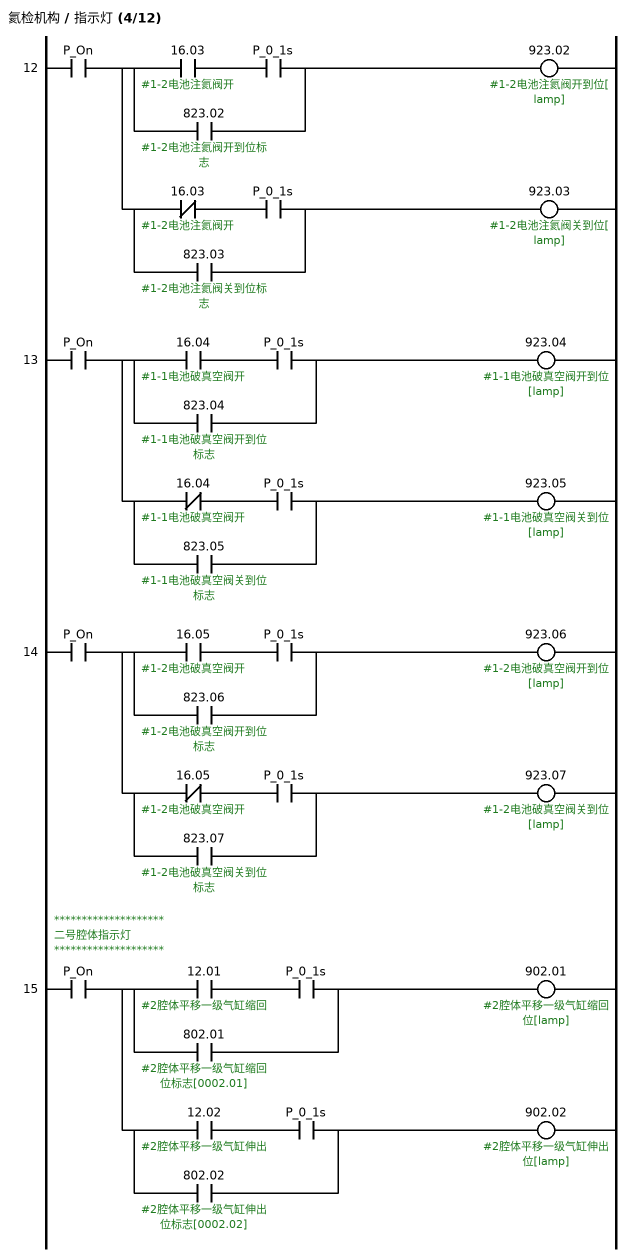
; [picture p360: 氦检机构 / 指示灯, rungs 12-15]
; rung 12
LD P_On
OUT TR0
LD 16.03  ; #1-2电池注氦阀开
AND P_0_1s
OR 823.02  ; #1-2电池注氦阀开到位标志
ANDLD
OUT 923.02  ; #1-2电池注氦阀开到位[lamp]
LD TR0
LDNOT 16.03  ; #1-2电池注氦阀开
AND P_0_1s
OR 823.03  ; #1-2电池注氦阀关到位标志
ANDLD
OUT 923.03  ; #1-2电池注氦阀关到位[lamp]
; rung 13
LD P_On
OUT TR0
LD 16.04  ; #1-1电池破真空阀开
AND P_0_1s
OR 823.04  ; #1-1电池破真空阀开到位标志
ANDLD
OUT 923.04  ; #1-1电池破真空阀开到位[lamp]
LD TR0
LDNOT 16.04  ; #1-1电池破真空阀开
AND P_0_1s
OR 823.05  ; #1-1电池破真空阀关到位标志
ANDLD
OUT 923.05  ; #1-1电池破真空阀关到位[lamp]
; rung 14
LD P_On
OUT TR0
LD 16.05  ; #1-2电池破真空阀开
AND P_0_1s
OR 823.06  ; #1-2电池破真空阀开到位标志
ANDLD
OUT 923.06  ; #1-2电池破真空阀开到位[lamp]
LD TR0
LDNOT 16.05  ; #1-2电池破真空阀开
AND P_0_1s
OR 823.07  ; #1-2电池破真空阀关到位标志
ANDLD
OUT 923.07  ; #1-2电池破真空阀关到位[lamp]
; rung 15: ******************** / 二号腔体指示灯 / ********************
LD P_On
OUT TR0
LD 12.01  ; #2腔体平移一级气缸缩回
AND P_0_1s
OR 802.01  ; #2腔体平移一级气缸缩回位标志[0002.01]
ANDLD
OUT 902.01  ; #2腔体平移一级气缸缩回位[lamp]
LD TR0
LD 12.02  ; #2腔体平移一级气缸伸出
AND P_0_1s
OR 802.02  ; #2腔体平移一级气缸伸出位标志[0002.02]
ANDLD
OUT 902.02  ; #2腔体平移一级气缸伸出位[lamp]

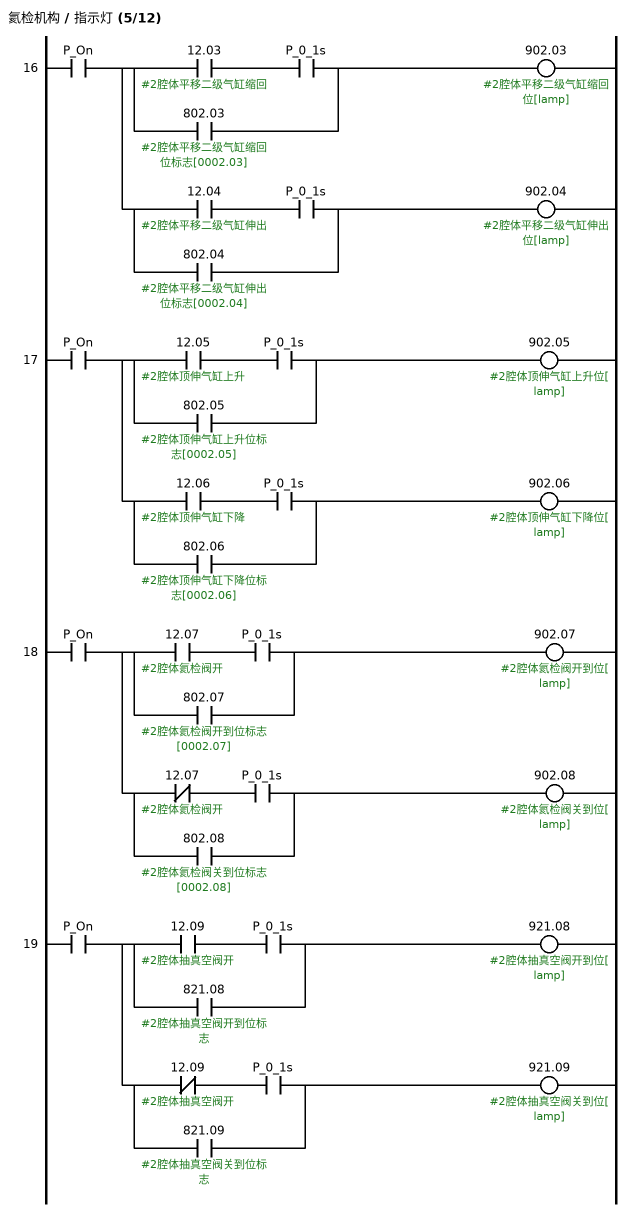
; rung 16
LD P_On
OUT TR0
LD 12.03  ; #2腔体平移二级气缸缩回
AND P_0_1s
OR 802.03  ; #2腔体平移二级气缸缩回位标志[0002.03]
ANDLD
OUT 902.03  ; #2腔体平移二级气缸缩回位[lamp]
LD TR0
LD 12.04  ; #2腔体平移二级气缸伸出
AND P_0_1s
OR 802.04  ; #2腔体平移二级气缸伸出位标志[0002.04]
ANDLD
OUT 902.04  ; #2腔体平移二级气缸伸出位[lamp]
; rung 17
LD P_On
OUT TR0
LD 12.05  ; #2腔体顶伸气缸上升
AND P_0_1s
OR 802.05  ; #2腔体顶伸气缸上升位标志[0002.05]
ANDLD
OUT 902.05  ; #2腔体顶伸气缸上升位[lamp]
LD TR0
LD 12.06  ; #2腔体顶伸气缸下降
AND P_0_1s
OR 802.06  ; #2腔体顶伸气缸下降位标志[0002.06]
ANDLD
OUT 902.06  ; #2腔体顶伸气缸下降位[lamp]
; rung 18
LD P_On
OUT TR0
LD 12.07  ; #2腔体氦检阀开
AND P_0_1s
OR 802.07  ; #2腔体氦检阀开到位标志[0002.07]
ANDLD
OUT 902.07  ; #2腔体氦检阀开到位[lamp]
LD TR0
LDNOT 12.07  ; #2腔体氦检阀开
AND P_0_1s
OR 802.08  ; #2腔体氦检阀关到位标志[0002.08]
ANDLD
OUT 902.08  ; #2腔体氦检阀关到位[lamp]
; rung 19
LD P_On
OUT TR0
LD 12.09  ; #2腔体抽真空阀开
AND P_0_1s
OR 821.08  ; #2腔体抽真空阀开到位标志
ANDLD
OUT 921.08  ; #2腔体抽真空阀开到位[lamp]
LD TR0
LDNOT 12.09  ; #2腔体抽真空阀开
AND P_0_1s
OR 821.09  ; #2腔体抽真空阀关到位标志
ANDLD
OUT 921.09  ; #2腔体抽真空阀关到位[lamp]

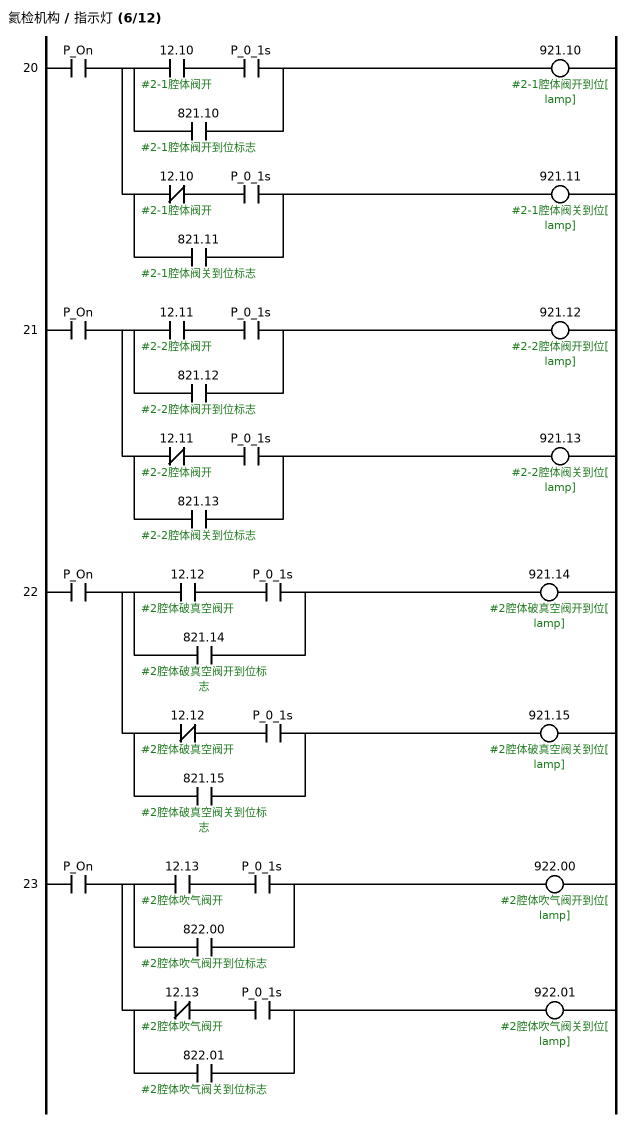
; rung 20
LD P_On
OUT TR0
LD 12.10  ; #2-1腔体阀开
AND P_0_1s
OR 821.10  ; #2-1腔体阀开到位标志
ANDLD
OUT 921.10  ; #2-1腔体阀开到位[lamp]
LD TR0
LDNOT 12.10  ; #2-1腔体阀开
AND P_0_1s
OR 821.11  ; #2-1腔体阀关到位标志
ANDLD
OUT 921.11  ; #2-1腔体阀关到位[lamp]
; rung 21
LD P_On
OUT TR0
LD 12.11  ; #2-2腔体阀开
AND P_0_1s
OR 821.12  ; #2-2腔体阀开到位标志
ANDLD
OUT 921.12  ; #2-2腔体阀开到位[lamp]
LD TR0
LDNOT 12.11  ; #2-2腔体阀开
AND P_0_1s
OR 821.13  ; #2-2腔体阀关到位标志
ANDLD
OUT 921.13  ; #2-2腔体阀关到位[lamp]
; rung 22
LD P_On
OUT TR0
LD 12.12  ; #2腔体破真空阀开
AND P_0_1s
OR 821.14  ; #2腔体破真空阀开到位标志
ANDLD
OUT 921.14  ; #2腔体破真空阀开到位[lamp]
LD TR0
LDNOT 12.12  ; #2腔体破真空阀开
AND P_0_1s
OR 821.15  ; #2腔体破真空阀关到位标志
ANDLD
OUT 921.15  ; #2腔体破真空阀关到位[lamp]
; rung 23
LD P_On
OUT TR0
LD 12.13  ; #2腔体吹气阀开
AND P_0_1s
OR 822.00  ; #2腔体吹气阀开到位标志
ANDLD
OUT 922.00  ; #2腔体吹气阀开到位[lamp]
LD TR0
LDNOT 12.13  ; #2腔体吹气阀开
AND P_0_1s
OR 822.01  ; #2腔体吹气阀关到位标志
ANDLD
OUT 922.01  ; #2腔体吹气阀关到位[lamp]

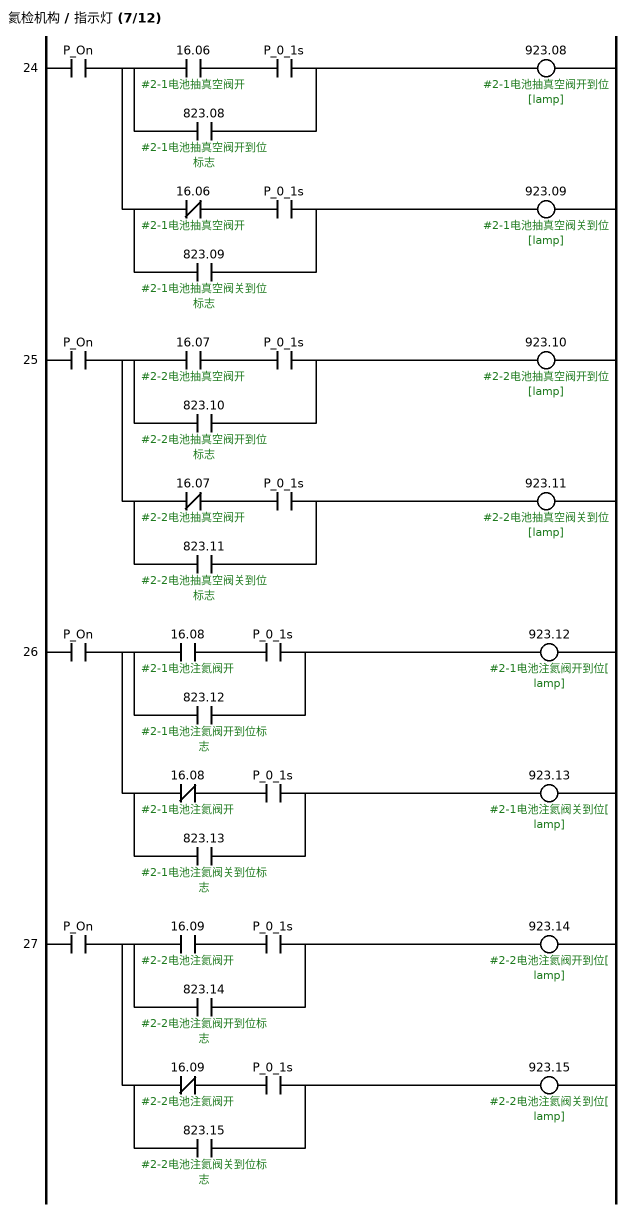
; rung 24
LD P_On
OUT TR0
LD 16.06  ; #2-1电池抽真空阀开
AND P_0_1s
OR 823.08  ; #2-1电池抽真空阀开到位标志
ANDLD
OUT 923.08  ; #2-1电池抽真空阀开到位[lamp]
LD TR0
LDNOT 16.06  ; #2-1电池抽真空阀开
AND P_0_1s
OR 823.09  ; #2-1电池抽真空阀关到位标志
ANDLD
OUT 923.09  ; #2-1电池抽真空阀关到位[lamp]
; rung 25
LD P_On
OUT TR0
LD 16.07  ; #2-2电池抽真空阀开
AND P_0_1s
OR 823.10  ; #2-2电池抽真空阀开到位标志
ANDLD
OUT 923.10  ; #2-2电池抽真空阀开到位[lamp]
LD TR0
LDNOT 16.07  ; #2-2电池抽真空阀开
AND P_0_1s
OR 823.11  ; #2-2电池抽真空阀关到位标志
ANDLD
OUT 923.11  ; #2-2电池抽真空阀关到位[lamp]
; rung 26
LD P_On
OUT TR0
LD 16.08  ; #2-1电池注氦阀开
AND P_0_1s
OR 823.12  ; #2-1电池注氦阀开到位标志
ANDLD
OUT 923.12  ; #2-1电池注氦阀开到位[lamp]
LD TR0
LDNOT 16.08  ; #2-1电池注氦阀开
AND P_0_1s
OR 823.13  ; #2-1电池注氦阀关到位标志
ANDLD
OUT 923.13  ; #2-1电池注氦阀关到位[lamp]
; rung 27
LD P_On
OUT TR0
LD 16.09  ; #2-2电池注氦阀开
AND P_0_1s
OR 823.14  ; #2-2电池注氦阀开到位标志
ANDLD
OUT 923.14  ; #2-2电池注氦阀开到位[lamp]
LD TR0
LDNOT 16.09  ; #2-2电池注氦阀开
AND P_0_1s
OR 823.15  ; #2-2电池注氦阀关到位标志
ANDLD
OUT 923.15  ; #2-2电池注氦阀关到位[lamp]

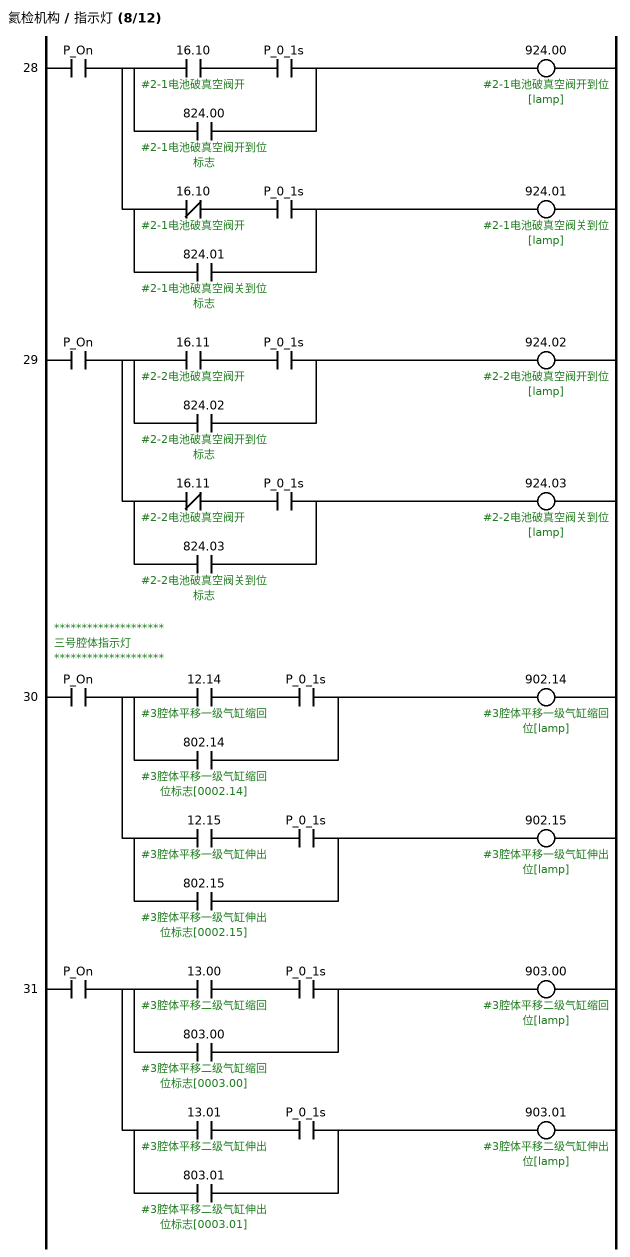
; rung 28
LD P_On
OUT TR0
LD 16.10  ; #2-1电池破真空阀开
AND P_0_1s
OR 824.00  ; #2-1电池破真空阀开到位标志
ANDLD
OUT 924.00  ; #2-1电池破真空阀开到位[lamp]
LD TR0
LDNOT 16.10  ; #2-1电池破真空阀开
AND P_0_1s
OR 824.01  ; #2-1电池破真空阀关到位标志
ANDLD
OUT 924.01  ; #2-1电池破真空阀关到位[lamp]
; rung 29
LD P_On
OUT TR0
LD 16.11  ; #2-2电池破真空阀开
AND P_0_1s
OR 824.02  ; #2-2电池破真空阀开到位标志
ANDLD
OUT 924.02  ; #2-2电池破真空阀开到位[lamp]
LD TR0
LDNOT 16.11  ; #2-2电池破真空阀开
AND P_0_1s
OR 824.03  ; #2-2电池破真空阀关到位标志
ANDLD
OUT 924.03  ; #2-2电池破真空阀关到位[lamp]
; rung 30: ******************** / 三号腔体指示灯 / ********************
LD P_On
OUT TR0
LD 12.14  ; #3腔体平移一级气缸缩回
AND P_0_1s
OR 802.14  ; #3腔体平移一级气缸缩回位标志[0002.14]
ANDLD
OUT 902.14  ; #3腔体平移一级气缸缩回位[lamp]
LD TR0
LD 12.15  ; #3腔体平移一级气缸伸出
AND P_0_1s
OR 802.15  ; #3腔体平移一级气缸伸出位标志[0002.15]
ANDLD
OUT 902.15  ; #3腔体平移一级气缸伸出位[lamp]
; rung 31
LD P_On
OUT TR0
LD 13.00  ; #3腔体平移二级气缸缩回
AND P_0_1s
OR 803.00  ; #3腔体平移二级气缸缩回位标志[0003.00]
ANDLD
OUT 903.00  ; #3腔体平移二级气缸缩回位[lamp]
LD TR0
LD 13.01  ; #3腔体平移二级气缸伸出
AND P_0_1s
OR 803.01  ; #3腔体平移二级气缸伸出位标志[0003.01]
ANDLD
OUT 903.01  ; #3腔体平移二级气缸伸出位[lamp]

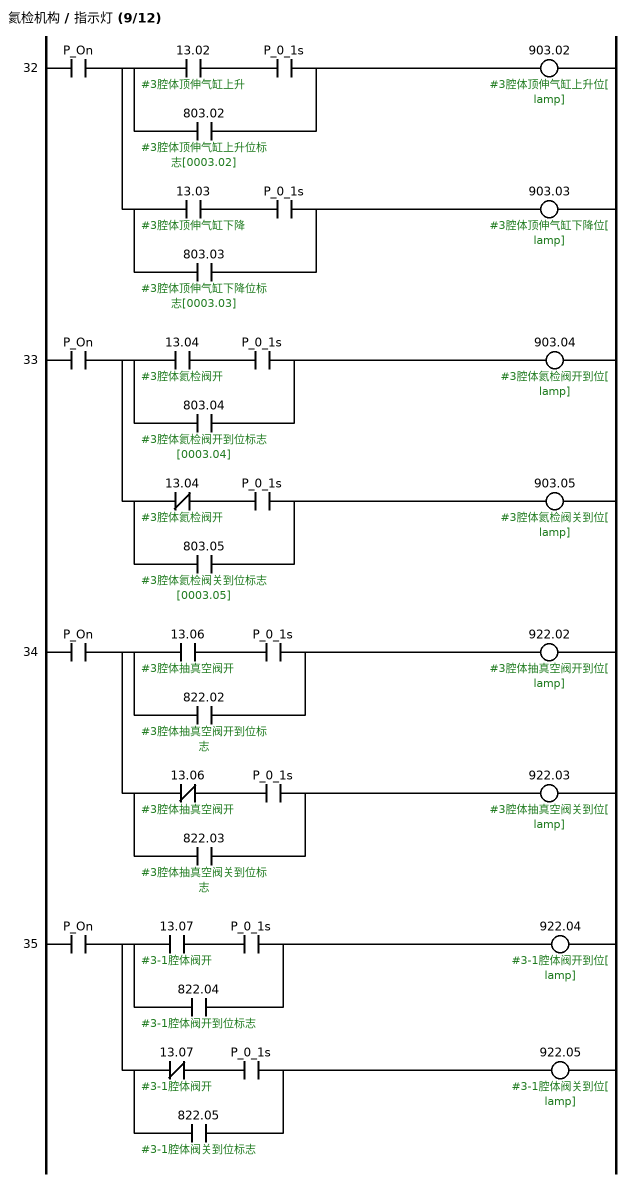
; rung 32
LD P_On
OUT TR0
LD 13.02  ; #3腔体顶伸气缸上升
AND P_0_1s
OR 803.02  ; #3腔体顶伸气缸上升位标志[0003.02]
ANDLD
OUT 903.02  ; #3腔体顶伸气缸上升位[lamp]
LD TR0
LD 13.03  ; #3腔体顶伸气缸下降
AND P_0_1s
OR 803.03  ; #3腔体顶伸气缸下降位标志[0003.03]
ANDLD
OUT 903.03  ; #3腔体顶伸气缸下降位[lamp]
; rung 33
LD P_On
OUT TR0
LD 13.04  ; #3腔体氦检阀开
AND P_0_1s
OR 803.04  ; #3腔体氦检阀开到位标志[0003.04]
ANDLD
OUT 903.04  ; #3腔体氦检阀开到位[lamp]
LD TR0
LDNOT 13.04  ; #3腔体氦检阀开
AND P_0_1s
OR 803.05  ; #3腔体氦检阀关到位标志[0003.05]
ANDLD
OUT 903.05  ; #3腔体氦检阀关到位[lamp]
; rung 34
LD P_On
OUT TR0
LD 13.06  ; #3腔体抽真空阀开
AND P_0_1s
OR 822.02  ; #3腔体抽真空阀开到位标志
ANDLD
OUT 922.02  ; #3腔体抽真空阀开到位[lamp]
LD TR0
LDNOT 13.06  ; #3腔体抽真空阀开
AND P_0_1s
OR 822.03  ; #3腔体抽真空阀关到位标志
ANDLD
OUT 922.03  ; #3腔体抽真空阀关到位[lamp]
; rung 35
LD P_On
OUT TR0
LD 13.07  ; #3-1腔体阀开
AND P_0_1s
OR 822.04  ; #3-1腔体阀开到位标志
ANDLD
OUT 922.04  ; #3-1腔体阀开到位[lamp]
LD TR0
LDNOT 13.07  ; #3-1腔体阀开
AND P_0_1s
OR 822.05  ; #3-1腔体阀关到位标志
ANDLD
OUT 922.05  ; #3-1腔体阀关到位[lamp]

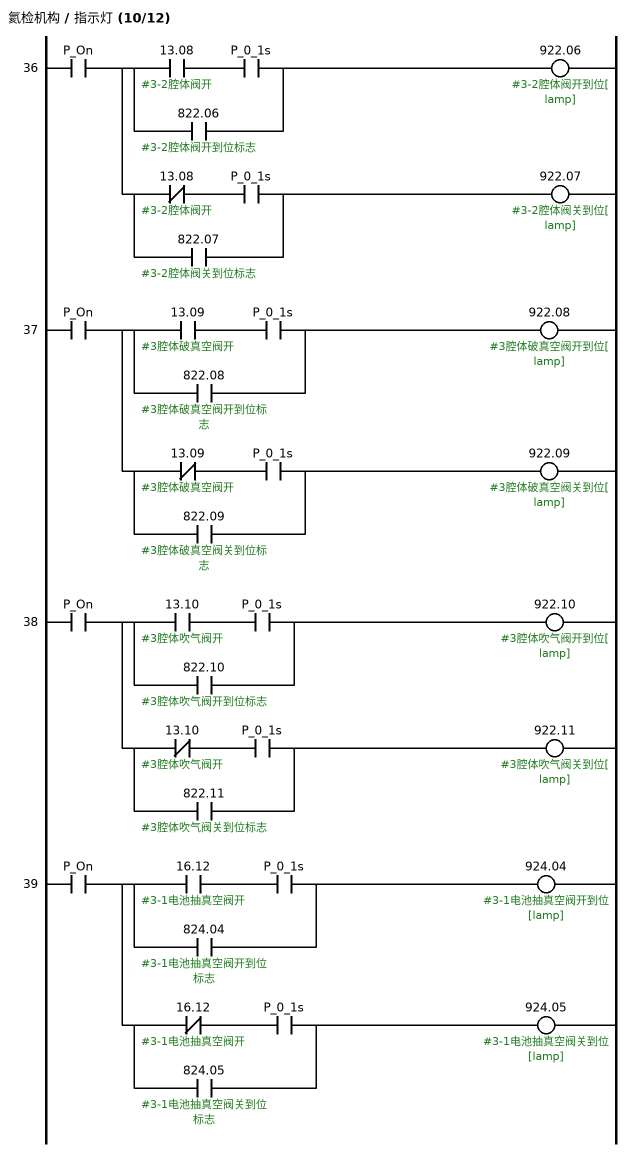
; rung 36
LD P_On
OUT TR0
LD 13.08  ; #3-2腔体阀开
AND P_0_1s
OR 822.06  ; #3-2腔体阀开到位标志
ANDLD
OUT 922.06  ; #3-2腔体阀开到位[lamp]
LD TR0
LDNOT 13.08  ; #3-2腔体阀开
AND P_0_1s
OR 822.07  ; #3-2腔体阀关到位标志
ANDLD
OUT 922.07  ; #3-2腔体阀关到位[lamp]
; rung 37
LD P_On
OUT TR0
LD 13.09  ; #3腔体破真空阀开
AND P_0_1s
OR 822.08  ; #3腔体破真空阀开到位标志
ANDLD
OUT 922.08  ; #3腔体破真空阀开到位[lamp]
LD TR0
LDNOT 13.09  ; #3腔体破真空阀开
AND P_0_1s
OR 822.09  ; #3腔体破真空阀关到位标志
ANDLD
OUT 922.09  ; #3腔体破真空阀关到位[lamp]
; rung 38
LD P_On
OUT TR0
LD 13.10  ; #3腔体吹气阀开
AND P_0_1s
OR 822.10  ; #3腔体吹气阀开到位标志
ANDLD
OUT 922.10  ; #3腔体吹气阀开到位[lamp]
LD TR0
LDNOT 13.10  ; #3腔体吹气阀开
AND P_0_1s
OR 822.11  ; #3腔体吹气阀关到位标志
ANDLD
OUT 922.11  ; #3腔体吹气阀关到位[lamp]
; rung 39
LD P_On
OUT TR0
LD 16.12  ; #3-1电池抽真空阀开
AND P_0_1s
OR 824.04  ; #3-1电池抽真空阀开到位标志
ANDLD
OUT 924.04  ; #3-1电池抽真空阀开到位[lamp]
LD TR0
LDNOT 16.12  ; #3-1电池抽真空阀开
AND P_0_1s
OR 824.05  ; #3-1电池抽真空阀关到位标志
ANDLD
OUT 924.05  ; #3-1电池抽真空阀关到位[lamp]

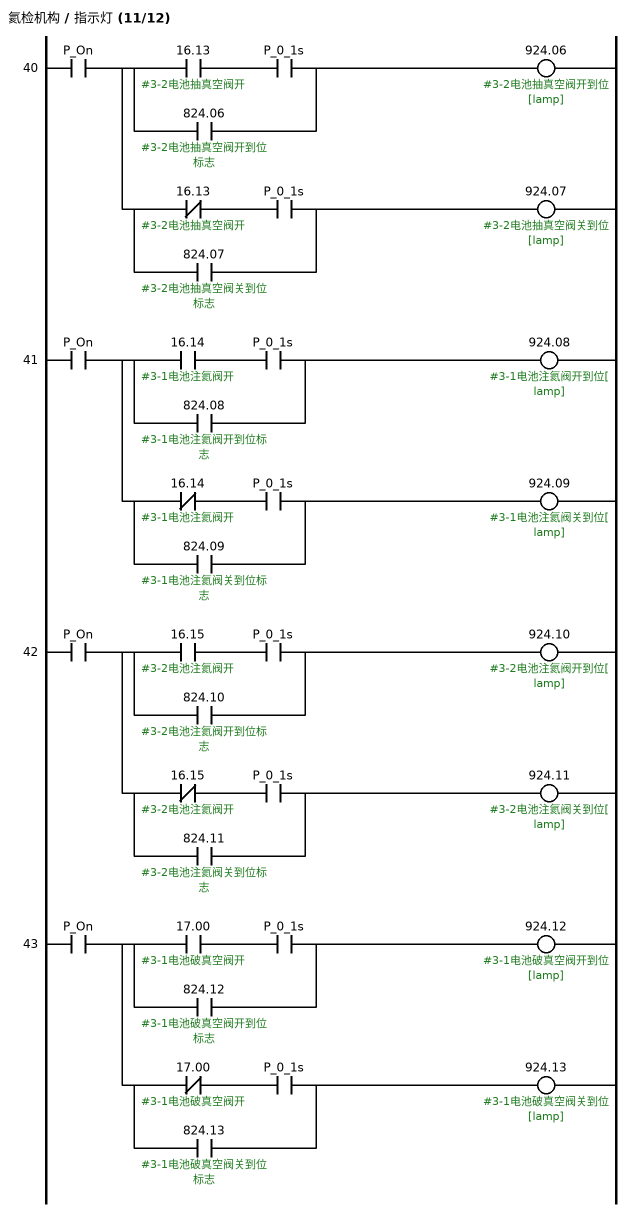
; rung 40
LD P_On
OUT TR0
LD 16.13  ; #3-2电池抽真空阀开
AND P_0_1s
OR 824.06  ; #3-2电池抽真空阀开到位标志
ANDLD
OUT 924.06  ; #3-2电池抽真空阀开到位[lamp]
LD TR0
LDNOT 16.13  ; #3-2电池抽真空阀开
AND P_0_1s
OR 824.07  ; #3-2电池抽真空阀关到位标志
ANDLD
OUT 924.07  ; #3-2电池抽真空阀关到位[lamp]
; rung 41
LD P_On
OUT TR0
LD 16.14  ; #3-1电池注氦阀开
AND P_0_1s
OR 824.08  ; #3-1电池注氦阀开到位标志
ANDLD
OUT 924.08  ; #3-1电池注氦阀开到位[lamp]
LD TR0
LDNOT 16.14  ; #3-1电池注氦阀开
AND P_0_1s
OR 824.09  ; #3-1电池注氦阀关到位标志
ANDLD
OUT 924.09  ; #3-1电池注氦阀关到位[lamp]
; rung 42
LD P_On
OUT TR0
LD 16.15  ; #3-2电池注氦阀开
AND P_0_1s
OR 824.10  ; #3-2电池注氦阀开到位标志
ANDLD
OUT 924.10  ; #3-2电池注氦阀开到位[lamp]
LD TR0
LDNOT 16.15  ; #3-2电池注氦阀开
AND P_0_1s
OR 824.11  ; #3-2电池注氦阀关到位标志
ANDLD
OUT 924.11  ; #3-2电池注氦阀关到位[lamp]
; rung 43
LD P_On
OUT TR0
LD 17.00  ; #3-1电池破真空阀开
AND P_0_1s
OR 824.12  ; #3-1电池破真空阀开到位标志
ANDLD
OUT 924.12  ; #3-1电池破真空阀开到位[lamp]
LD TR0
LDNOT 17.00  ; #3-1电池破真空阀开
AND P_0_1s
OR 824.13  ; #3-1电池破真空阀关到位标志
ANDLD
OUT 924.13  ; #3-1电池破真空阀关到位[lamp]

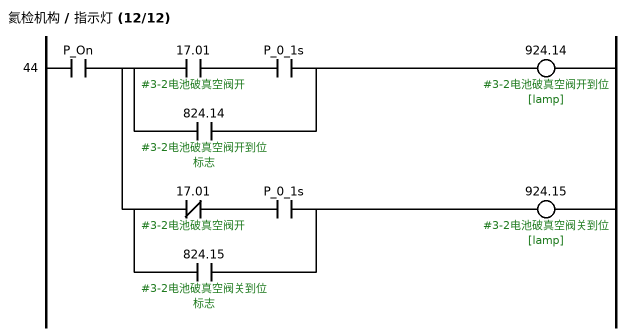
; rung 44
LD P_On
OUT TR0
LD 17.01  ; #3-2电池破真空阀开
AND P_0_1s
OR 824.14  ; #3-2电池破真空阀开到位标志
ANDLD
OUT 924.14  ; #3-2电池破真空阀开到位[lamp]
LD TR0
LDNOT 17.01  ; #3-2电池破真空阀开
AND P_0_1s
OR 824.15  ; #3-2电池破真空阀关到位标志
ANDLD
OUT 924.15  ; #3-2电池破真空阀关到位[lamp]

### Section 外部输出

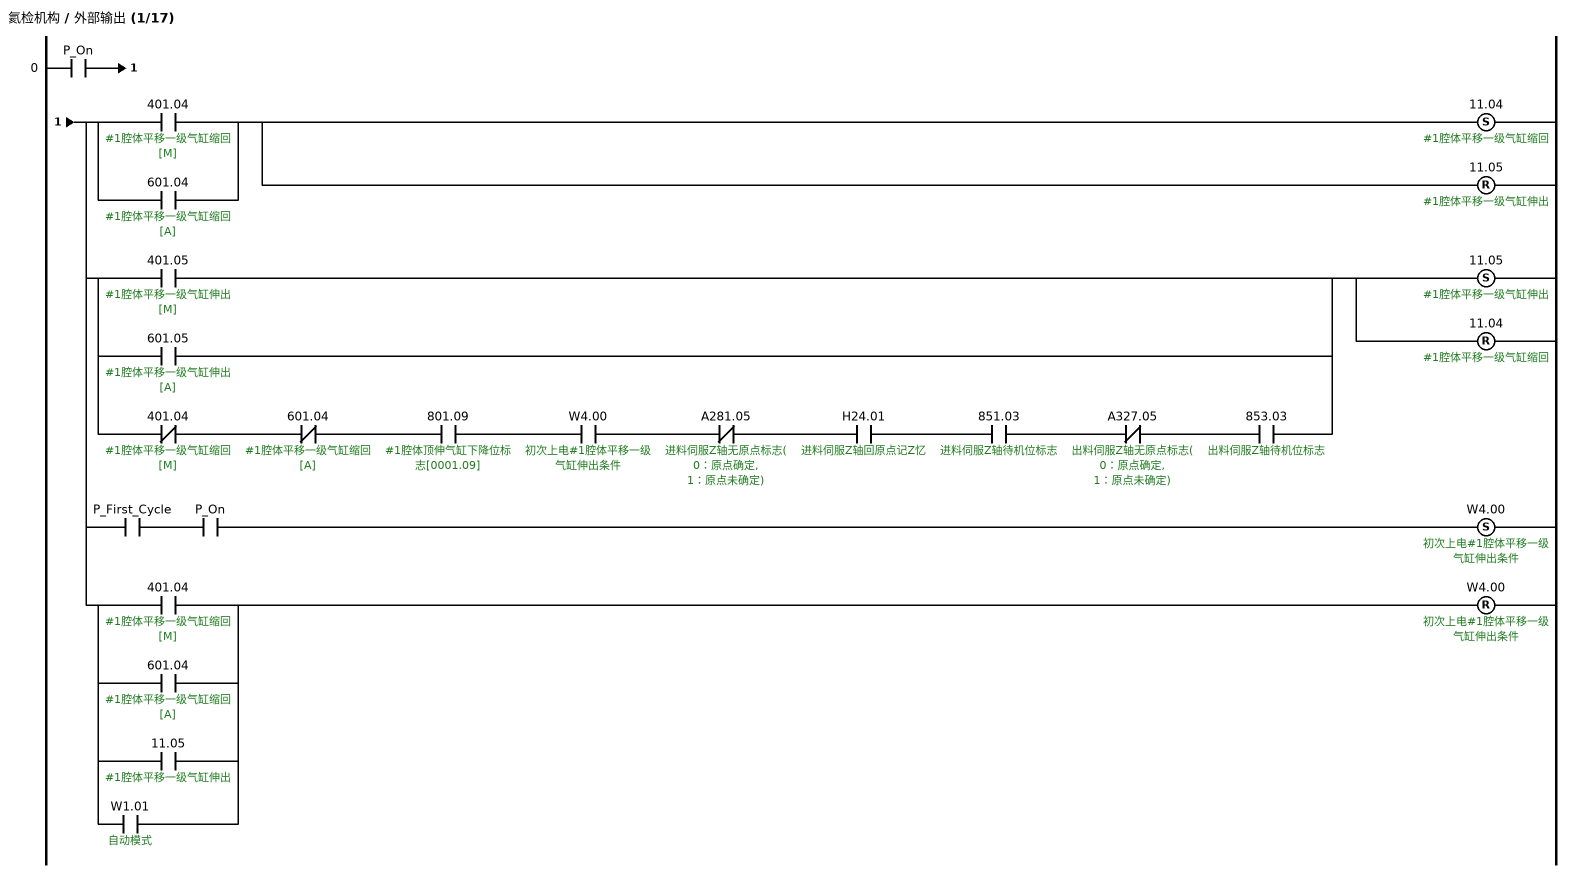
; rung 0
LD P_On
OUT TR0
LD 401.04  ; #1腔体平移一级气缸缩回[M]
OR 601.04  ; #1腔体平移一级气缸缩回[A]
ANDLD
SET 11.04  ; #1腔体平移一级气缸缩回
RSET 11.05  ; #1腔体平移一级气缸伸出
LD TR0
LD 401.05  ; #1腔体平移一级气缸伸出[M]
OR 601.05  ; #1腔体平移一级气缸伸出[A]
LDNOT 401.04  ; #1腔体平移一级气缸缩回[M]
ANDNOT 601.04  ; #1腔体平移一级气缸缩回[A]
AND 801.09  ; #1腔体顶伸气缸下降位标志[0001.09]
AND W4.00  ; 初次上电#1腔体平移一级气缸伸出条件
ANDNOT A281.05  ; 进料伺服Z轴无原点标志(0：原点确定,1：原点未确定)
AND H24.01  ; 进料伺服Z轴回原点记Z忆
AND 851.03  ; 进料伺服Z轴待机位标志
ANDNOT A327.05  ; 出料伺服Z轴无原点标志(0：原点确定,1：原点未确定)
AND 853.03  ; 出料伺服Z轴待机位标志
ORLD
ANDLD
SET 11.05  ; #1腔体平移一级气缸伸出
RSET 11.04  ; #1腔体平移一级气缸缩回
LD TR0
AND P_First_Cycle
AND P_On
SET W4.00  ; 初次上电#1腔体平移一级气缸伸出条件
LD TR0
LD 401.04  ; #1腔体平移一级气缸缩回[M]
OR 601.04  ; #1腔体平移一级气缸缩回[A]
OR 11.05  ; #1腔体平移一级气缸伸出
OR W1.01  ; 自动模式
ANDLD
RSET W4.00  ; 初次上电#1腔体平移一级气缸伸出条件

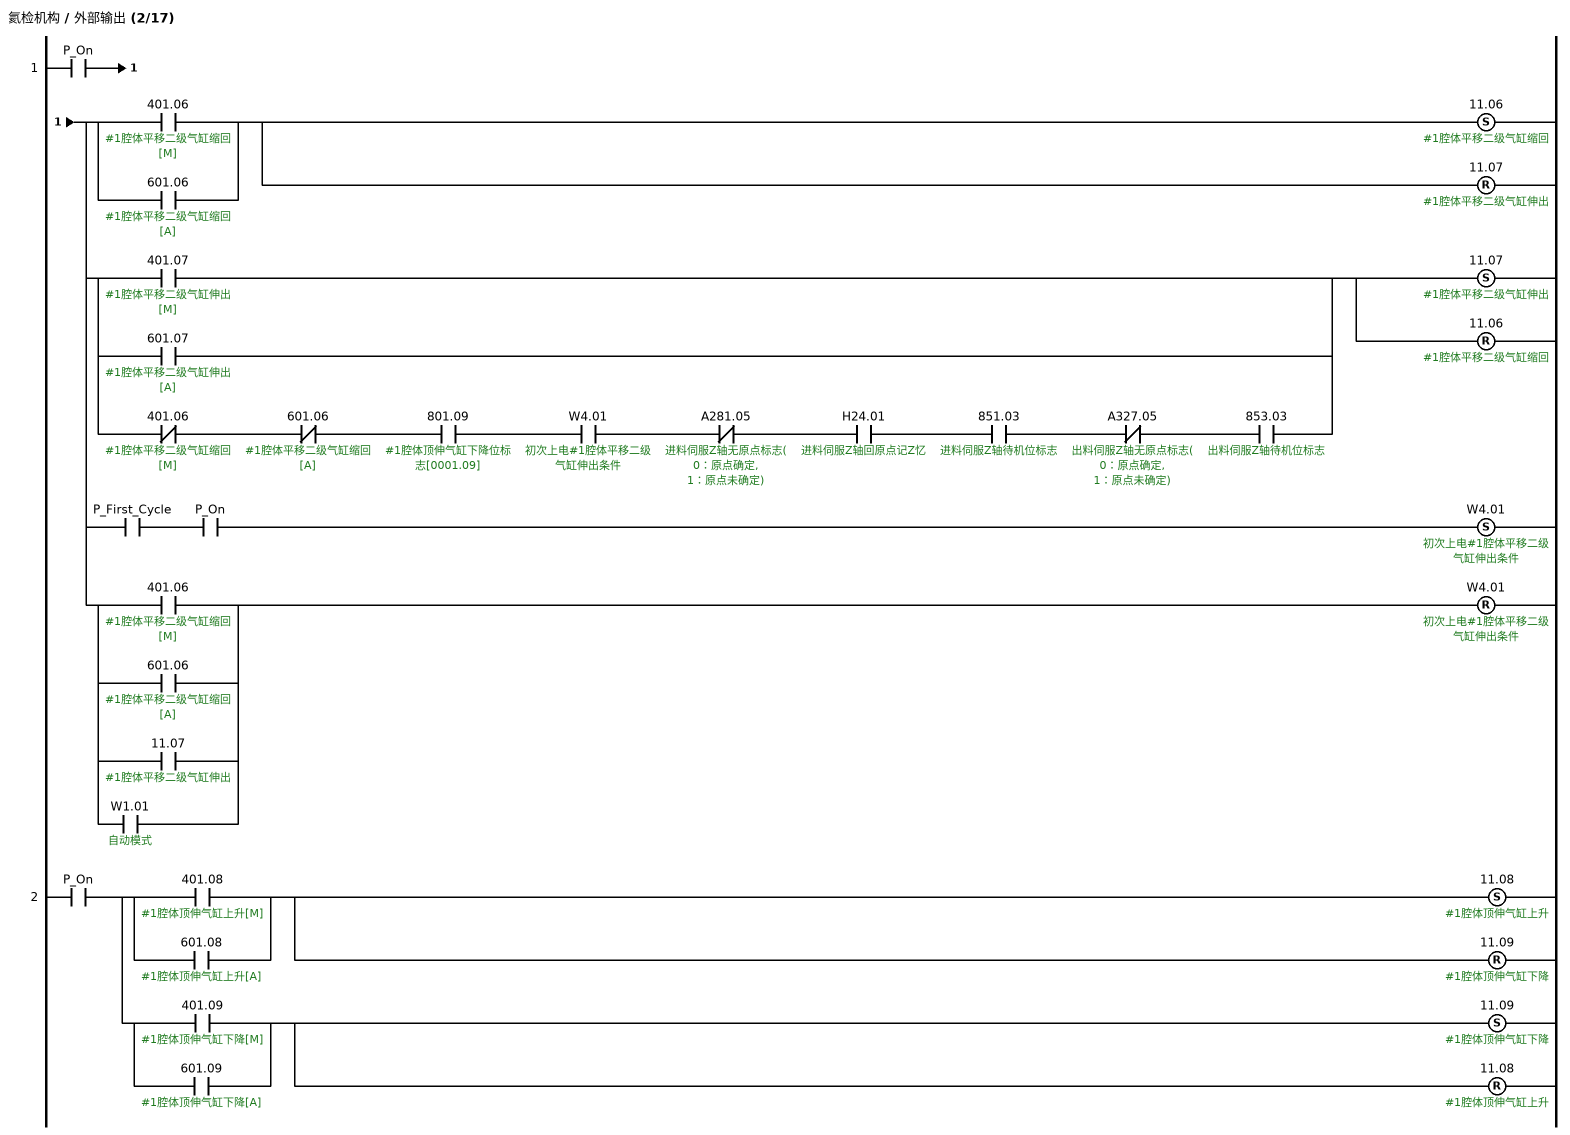
; rung 1
LD P_On
OUT TR0
LD 401.06  ; #1腔体平移二级气缸缩回[M]
OR 601.06  ; #1腔体平移二级气缸缩回[A]
ANDLD
SET 11.06  ; #1腔体平移二级气缸缩回
RSET 11.07  ; #1腔体平移二级气缸伸出
LD TR0
LD 401.07  ; #1腔体平移二级气缸伸出[M]
OR 601.07  ; #1腔体平移二级气缸伸出[A]
LDNOT 401.06  ; #1腔体平移二级气缸缩回[M]
ANDNOT 601.06  ; #1腔体平移二级气缸缩回[A]
AND 801.09  ; #1腔体顶伸气缸下降位标志[0001.09]
AND W4.01  ; 初次上电#1腔体平移二级气缸伸出条件
ANDNOT A281.05  ; 进料伺服Z轴无原点标志(0：原点确定,1：原点未确定)
AND H24.01  ; 进料伺服Z轴回原点记Z忆
AND 851.03  ; 进料伺服Z轴待机位标志
ANDNOT A327.05  ; 出料伺服Z轴无原点标志(0：原点确定,1：原点未确定)
AND 853.03  ; 出料伺服Z轴待机位标志
ORLD
ANDLD
SET 11.07  ; #1腔体平移二级气缸伸出
RSET 11.06  ; #1腔体平移二级气缸缩回
LD TR0
AND P_First_Cycle
AND P_On
SET W4.01  ; 初次上电#1腔体平移二级气缸伸出条件
LD TR0
LD 401.06  ; #1腔体平移二级气缸缩回[M]
OR 601.06  ; #1腔体平移二级气缸缩回[A]
OR 11.07  ; #1腔体平移二级气缸伸出
OR W1.01  ; 自动模式
ANDLD
RSET W4.01  ; 初次上电#1腔体平移二级气缸伸出条件
; rung 2
LD P_On
OUT TR0
LD 401.08  ; #1腔体顶伸气缸上升[M]
OR 601.08  ; #1腔体顶伸气缸上升[A]
ANDLD
SET 11.08  ; #1腔体顶伸气缸上升
RSET 11.09  ; #1腔体顶伸气缸下降
LD TR0
LD 401.09  ; #1腔体顶伸气缸下降[M]
OR 601.09  ; #1腔体顶伸气缸下降[A]
ANDLD
SET 11.09  ; #1腔体顶伸气缸下降
RSET 11.08  ; #1腔体顶伸气缸上升

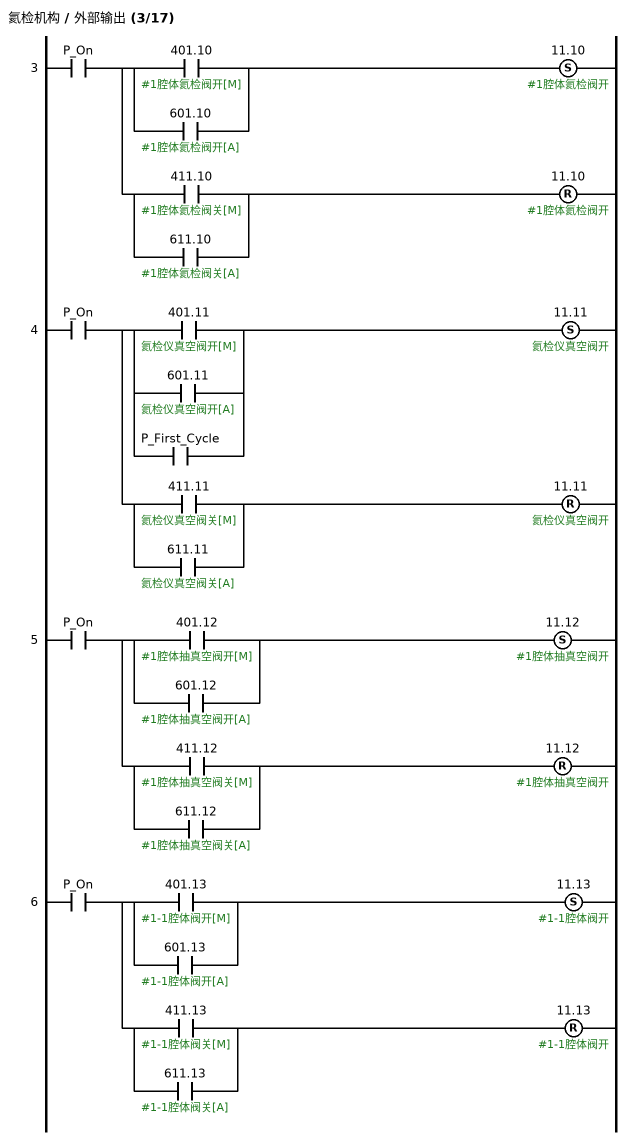
; rung 3
LD P_On
OUT TR0
LD 401.10  ; #1腔体氦检阀开[M]
OR 601.10  ; #1腔体氦检阀开[A]
ANDLD
SET 11.10  ; #1腔体氦检阀开
LD TR0
LD 411.10  ; #1腔体氦检阀关[M]
OR 611.10  ; #1腔体氦检阀关[A]
ANDLD
RSET 11.10  ; #1腔体氦检阀开
; rung 4
LD P_On
OUT TR0
LD 401.11  ; 氦检仪真空阀开[M]
OR 601.11  ; 氦检仪真空阀开[A]
OR P_First_Cycle  // 保证氦检仪开启时能将管路抽成真空状态
ANDLD
SET 11.11  ; 氦检仪真空阀开
LD TR0
LD 411.11  ; 氦检仪真空阀关[M]
OR 611.11  ; 氦检仪真空阀关[A]
ANDLD
RSET 11.11  ; 氦检仪真空阀开
; rung 5
LD P_On
OUT TR0
LD 401.12  ; #1腔体抽真空阀开[M]
OR 601.12  ; #1腔体抽真空阀开[A]
ANDLD
SET 11.12  ; #1腔体抽真空阀开
LD TR0
LD 411.12  ; #1腔体抽真空阀关[M]
OR 611.12  ; #1腔体抽真空阀关[A]
ANDLD
RSET 11.12  ; #1腔体抽真空阀开
; rung 6
LD P_On
OUT TR0
LD 401.13  ; #1-1腔体阀开[M]
OR 601.13  ; #1-1腔体阀开[A]
ANDLD
SET 11.13  ; #1-1腔体阀开
LD TR0
LD 411.13  ; #1-1腔体阀关[M]
OR 611.13  ; #1-1腔体阀关[A]
ANDLD
RSET 11.13  ; #1-1腔体阀开

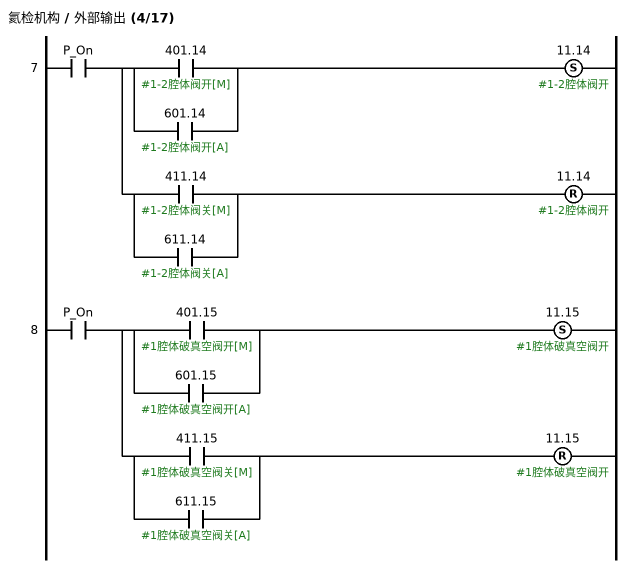
; rung 7
LD P_On
OUT TR0
LD 401.14  ; #1-2腔体阀开[M]
OR 601.14  ; #1-2腔体阀开[A]
ANDLD
SET 11.14  ; #1-2腔体阀开
LD TR0
LD 411.14  ; #1-2腔体阀关[M]
OR 611.14  ; #1-2腔体阀关[A]
ANDLD
RSET 11.14  ; #1-2腔体阀开
; rung 8
LD P_On
OUT TR0
LD 401.15  ; #1腔体破真空阀开[M]
OR 601.15  ; #1腔体破真空阀开[A]
ANDLD
SET 11.15  ; #1腔体破真空阀开
LD TR0
LD 411.15  ; #1腔体破真空阀关[M]
OR 611.15  ; #1腔体破真空阀关[A]
ANDLD
RSET 11.15  ; #1腔体破真空阀开

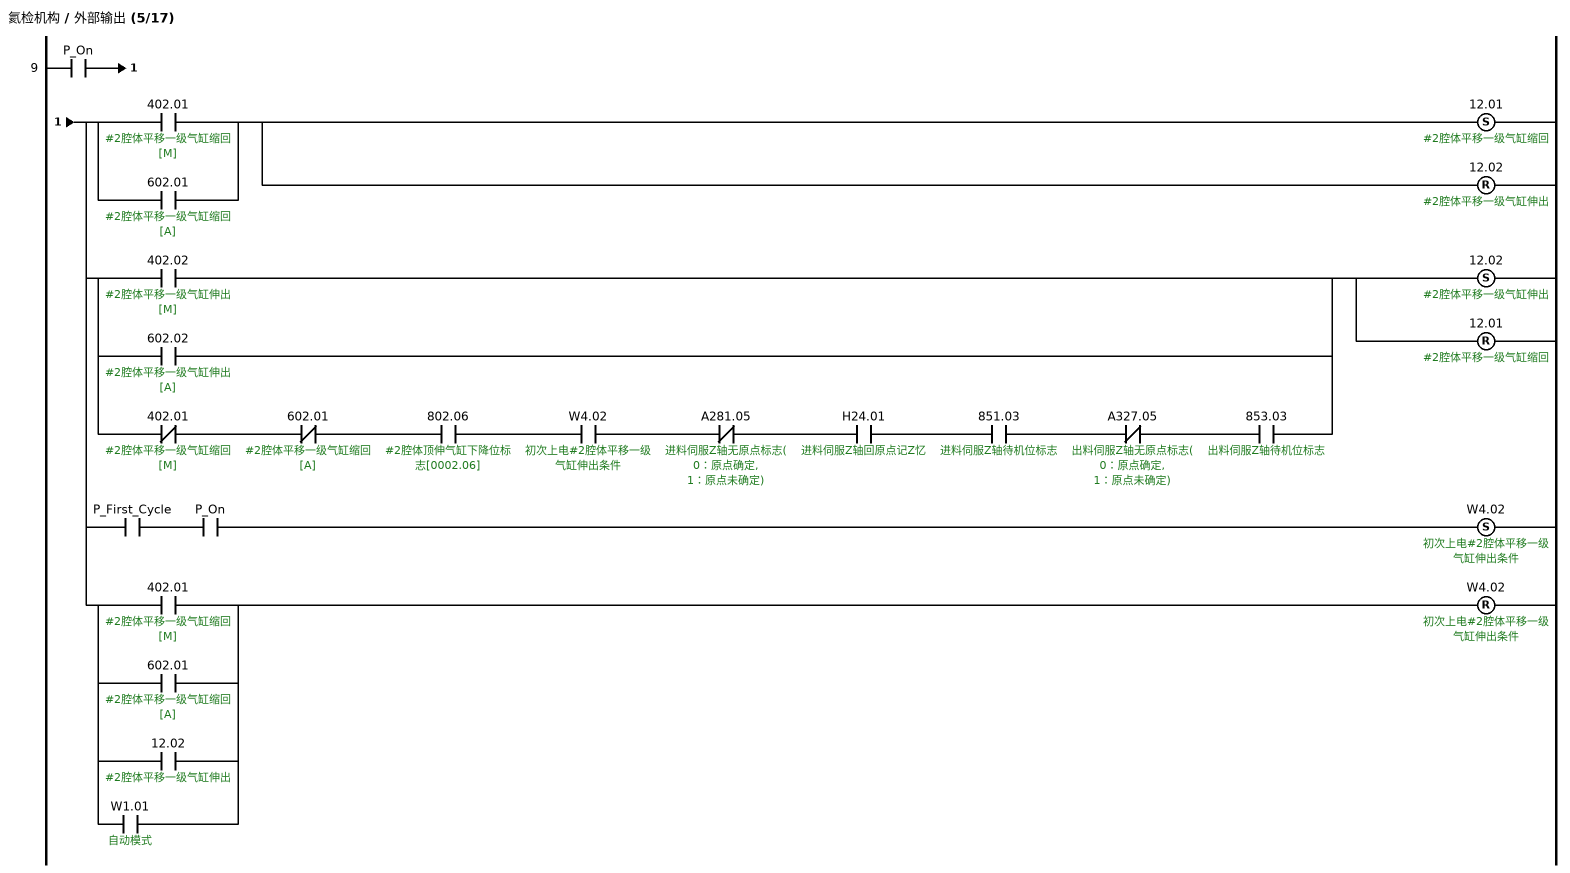
; rung 9
LD P_On
OUT TR0
LD 402.01  ; #2腔体平移一级气缸缩回[M]
OR 602.01  ; #2腔体平移一级气缸缩回[A]
ANDLD
SET 12.01  ; #2腔体平移一级气缸缩回
RSET 12.02  ; #2腔体平移一级气缸伸出
LD TR0
LD 402.02  ; #2腔体平移一级气缸伸出[M]
OR 602.02  ; #2腔体平移一级气缸伸出[A]
LDNOT 402.01  ; #2腔体平移一级气缸缩回[M]
ANDNOT 602.01  ; #2腔体平移一级气缸缩回[A]
AND 802.06  ; #2腔体顶伸气缸下降位标志[0002.06]
AND W4.02  ; 初次上电#2腔体平移一级气缸伸出条件
ANDNOT A281.05  ; 进料伺服Z轴无原点标志(0：原点确定,1：原点未确定)
AND H24.01  ; 进料伺服Z轴回原点记Z忆
AND 851.03  ; 进料伺服Z轴待机位标志
ANDNOT A327.05  ; 出料伺服Z轴无原点标志(0：原点确定,1：原点未确定)
AND 853.03  ; 出料伺服Z轴待机位标志
ORLD
ANDLD
SET 12.02  ; #2腔体平移一级气缸伸出
RSET 12.01  ; #2腔体平移一级气缸缩回
LD TR0
AND P_First_Cycle
AND P_On
SET W4.02  ; 初次上电#2腔体平移一级气缸伸出条件
LD TR0
LD 402.01  ; #2腔体平移一级气缸缩回[M]
OR 602.01  ; #2腔体平移一级气缸缩回[A]
OR 12.02  ; #2腔体平移一级气缸伸出
OR W1.01  ; 自动模式
ANDLD
RSET W4.02  ; 初次上电#2腔体平移一级气缸伸出条件

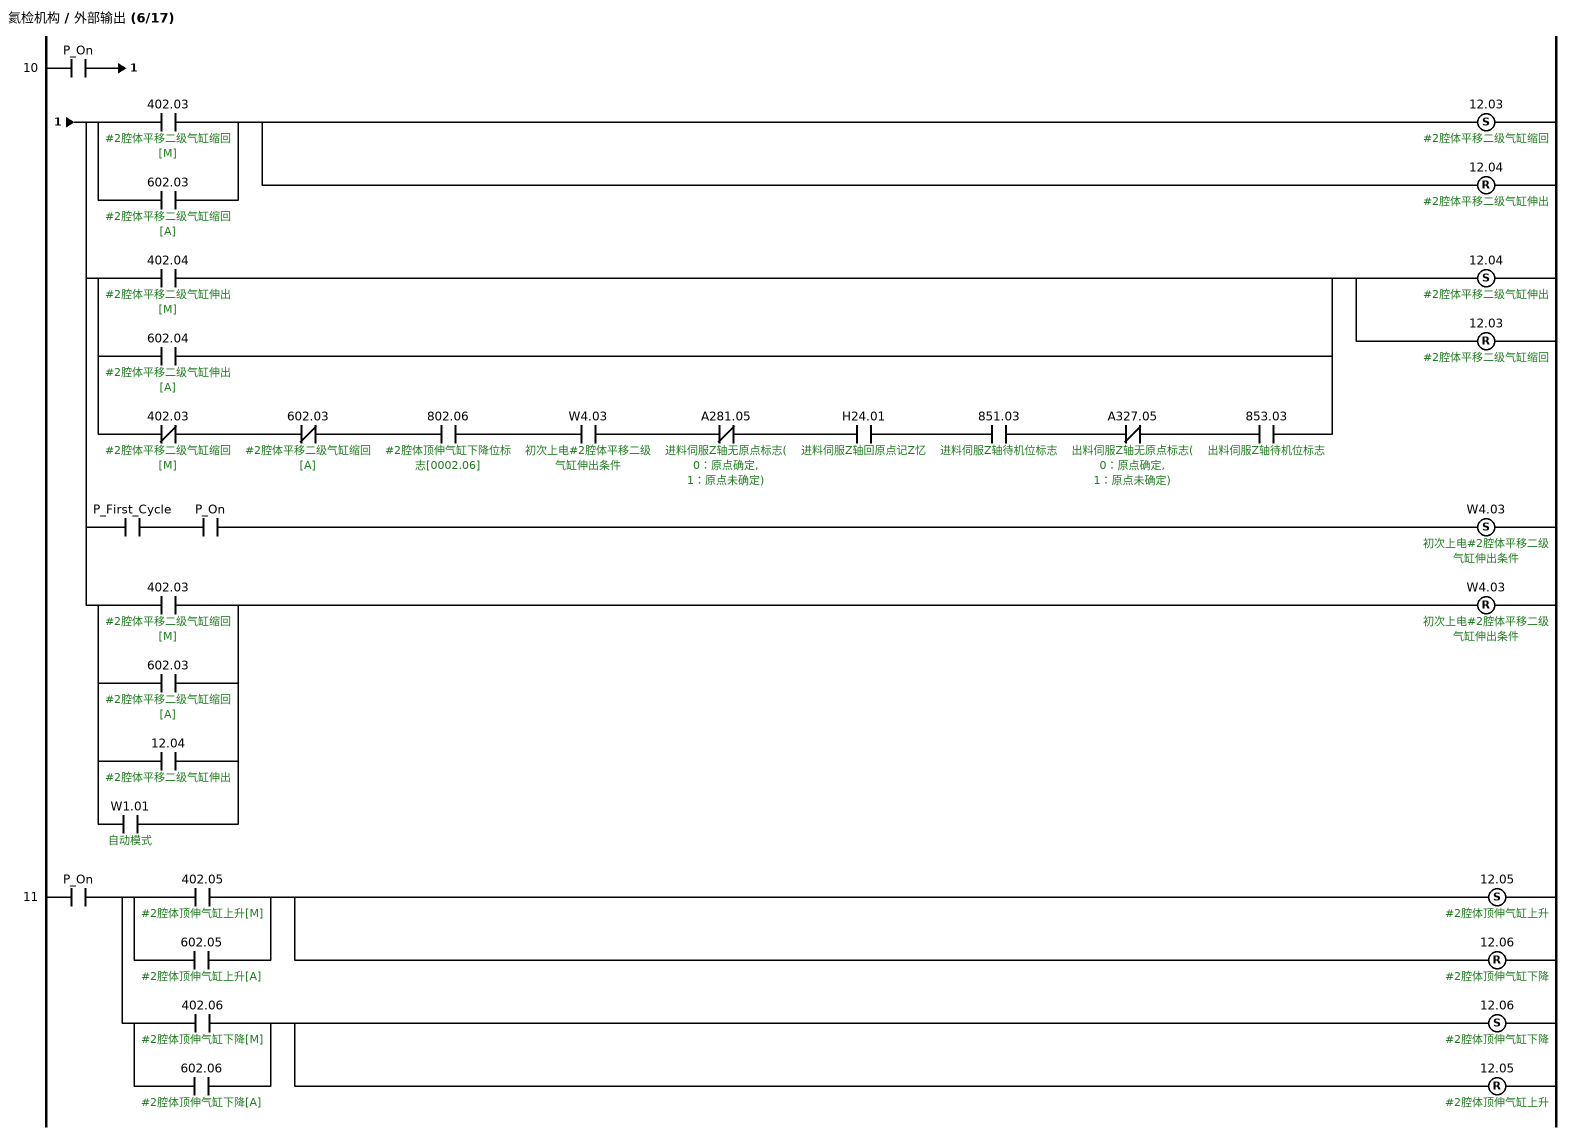
; rung 10
LD P_On
OUT TR0
LD 402.03  ; #2腔体平移二级气缸缩回[M]
OR 602.03  ; #2腔体平移二级气缸缩回[A]
ANDLD
SET 12.03  ; #2腔体平移二级气缸缩回
RSET 12.04  ; #2腔体平移二级气缸伸出
LD TR0
LD 402.04  ; #2腔体平移二级气缸伸出[M]
OR 602.04  ; #2腔体平移二级气缸伸出[A]
LDNOT 402.03  ; #2腔体平移二级气缸缩回[M]
ANDNOT 602.03  ; #2腔体平移二级气缸缩回[A]
AND 802.06  ; #2腔体顶伸气缸下降位标志[0002.06]
AND W4.03  ; 初次上电#2腔体平移二级气缸伸出条件
ANDNOT A281.05  ; 进料伺服Z轴无原点标志(0：原点确定,1：原点未确定)
AND H24.01  ; 进料伺服Z轴回原点记Z忆
AND 851.03  ; 进料伺服Z轴待机位标志
ANDNOT A327.05  ; 出料伺服Z轴无原点标志(0：原点确定,1：原点未确定)
AND 853.03  ; 出料伺服Z轴待机位标志
ORLD
ANDLD
SET 12.04  ; #2腔体平移二级气缸伸出
RSET 12.03  ; #2腔体平移二级气缸缩回
LD TR0
AND P_First_Cycle
AND P_On
SET W4.03  ; 初次上电#2腔体平移二级气缸伸出条件
LD TR0
LD 402.03  ; #2腔体平移二级气缸缩回[M]
OR 602.03  ; #2腔体平移二级气缸缩回[A]
OR 12.04  ; #2腔体平移二级气缸伸出
OR W1.01  ; 自动模式
ANDLD
RSET W4.03  ; 初次上电#2腔体平移二级气缸伸出条件
; rung 11
LD P_On
OUT TR0
LD 402.05  ; #2腔体顶伸气缸上升[M]
OR 602.05  ; #2腔体顶伸气缸上升[A]
ANDLD
SET 12.05  ; #2腔体顶伸气缸上升
RSET 12.06  ; #2腔体顶伸气缸下降
LD TR0
LD 402.06  ; #2腔体顶伸气缸下降[M]
OR 602.06  ; #2腔体顶伸气缸下降[A]
ANDLD
SET 12.06  ; #2腔体顶伸气缸下降
RSET 12.05  ; #2腔体顶伸气缸上升

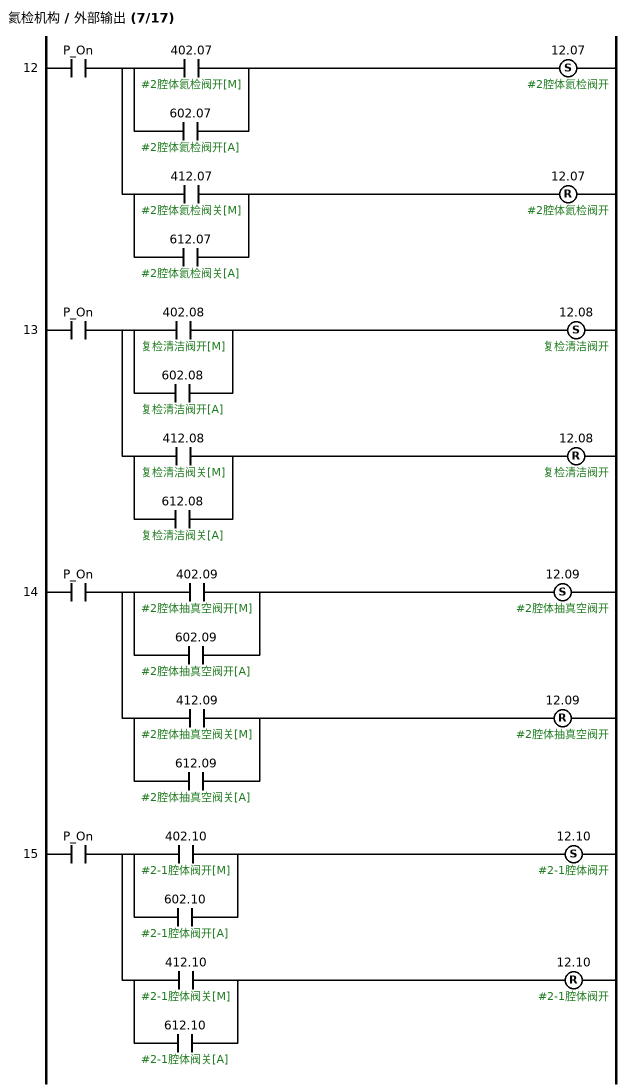
; rung 12
LD P_On
OUT TR0
LD 402.07  ; #2腔体氦检阀开[M]
OR 602.07  ; #2腔体氦检阀开[A]
ANDLD
SET 12.07  ; #2腔体氦检阀开
LD TR0
LD 412.07  ; #2腔体氦检阀关[M]
OR 612.07  ; #2腔体氦检阀关[A]
ANDLD
RSET 12.07  ; #2腔体氦检阀开
; rung 13
LD P_On
OUT TR0
LD 402.08  ; 复检清洁阀开[M]
OR 602.08  ; 复检清洁阀开[A]
ANDLD
SET 12.08  ; 复检清洁阀开
LD TR0
LD 412.08  ; 复检清洁阀关[M]
OR 612.08  ; 复检清洁阀关[A]
ANDLD
RSET 12.08  ; 复检清洁阀开
; rung 14
LD P_On
OUT TR0
LD 402.09  ; #2腔体抽真空阀开[M]
OR 602.09  ; #2腔体抽真空阀开[A]
ANDLD
SET 12.09  ; #2腔体抽真空阀开
LD TR0
LD 412.09  ; #2腔体抽真空阀关[M]
OR 612.09  ; #2腔体抽真空阀关[A]
ANDLD
RSET 12.09  ; #2腔体抽真空阀开
; rung 15
LD P_On
OUT TR0
LD 402.10  ; #2-1腔体阀开[M]
OR 602.10  ; #2-1腔体阀开[A]
ANDLD
SET 12.10  ; #2-1腔体阀开
LD TR0
LD 412.10  ; #2-1腔体阀关[M]
OR 612.10  ; #2-1腔体阀关[A]
ANDLD
RSET 12.10  ; #2-1腔体阀开

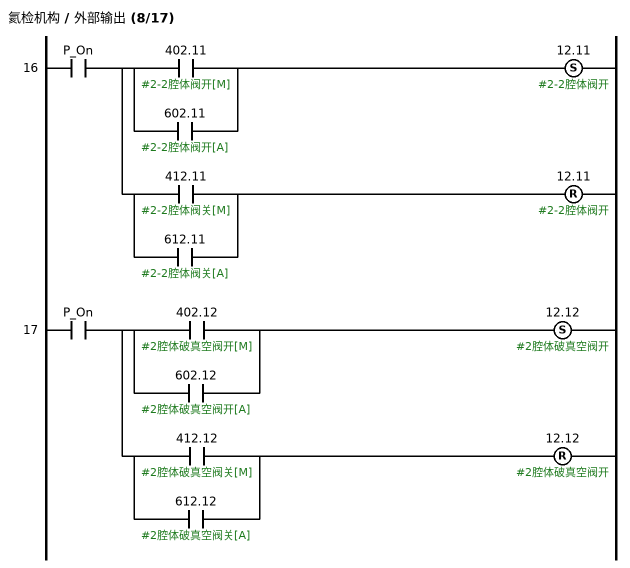
; rung 16
LD P_On
OUT TR0
LD 402.11  ; #2-2腔体阀开[M]
OR 602.11  ; #2-2腔体阀开[A]
ANDLD
SET 12.11  ; #2-2腔体阀开
LD TR0
LD 412.11  ; #2-2腔体阀关[M]
OR 612.11  ; #2-2腔体阀关[A]
ANDLD
RSET 12.11  ; #2-2腔体阀开
; rung 17
LD P_On
OUT TR0
LD 402.12  ; #2腔体破真空阀开[M]
OR 602.12  ; #2腔体破真空阀开[A]
ANDLD
SET 12.12  ; #2腔体破真空阀开
LD TR0
LD 412.12  ; #2腔体破真空阀关[M]
OR 612.12  ; #2腔体破真空阀关[A]
ANDLD
RSET 12.12  ; #2腔体破真空阀开

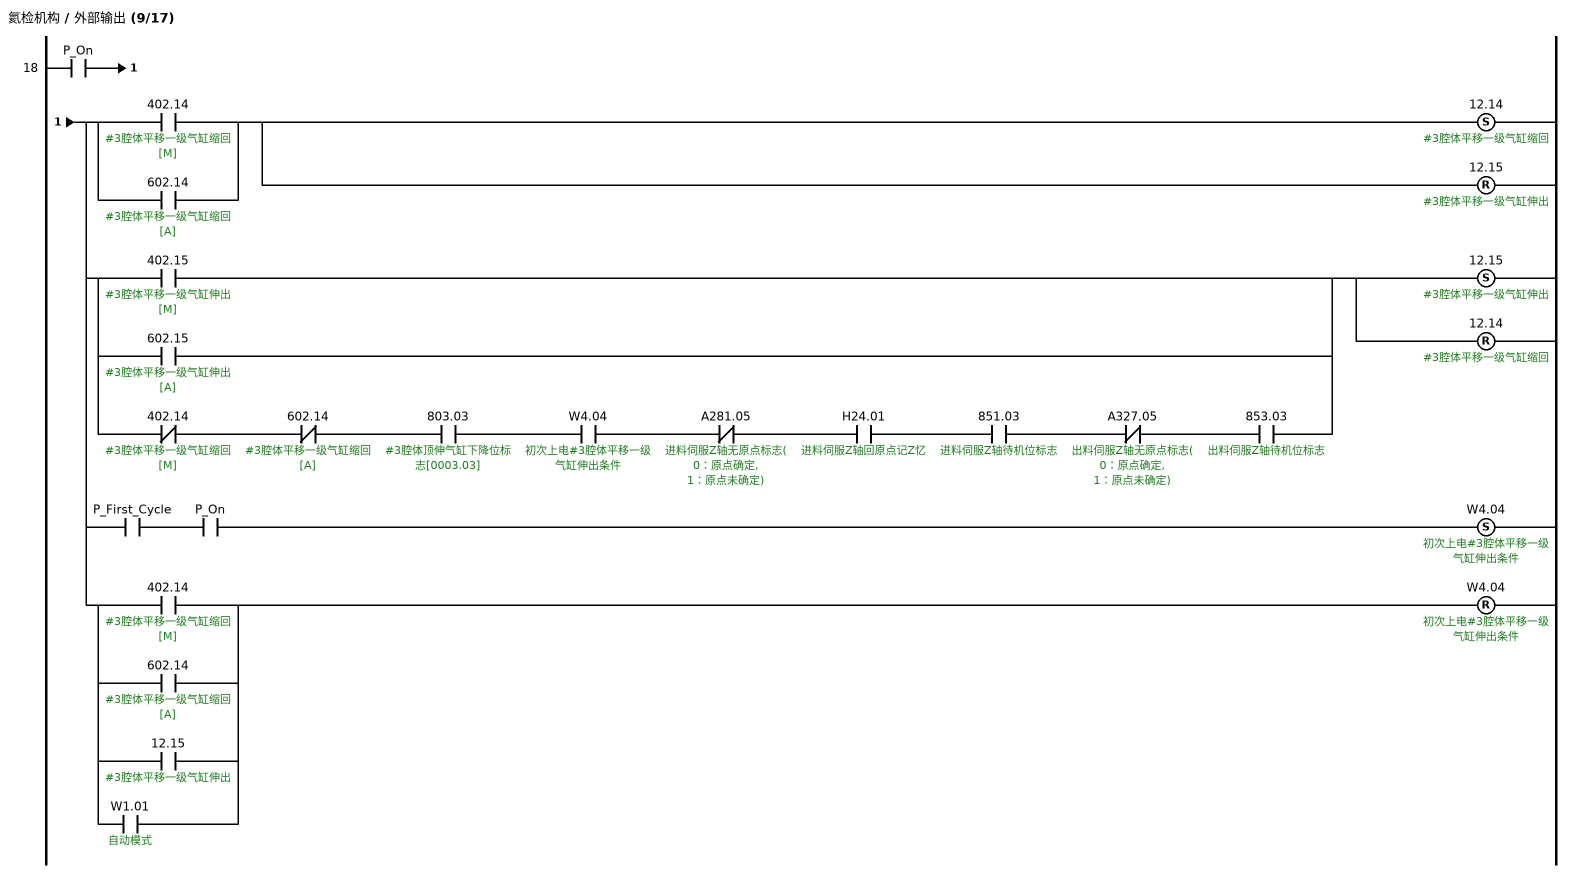
; rung 18
LD P_On
OUT TR0
LD 402.14  ; #3腔体平移一级气缸缩回[M]
OR 602.14  ; #3腔体平移一级气缸缩回[A]
ANDLD
SET 12.14  ; #3腔体平移一级气缸缩回
RSET 12.15  ; #3腔体平移一级气缸伸出
LD TR0
LD 402.15  ; #3腔体平移一级气缸伸出[M]
OR 602.15  ; #3腔体平移一级气缸伸出[A]
LDNOT 402.14  ; #3腔体平移一级气缸缩回[M]
ANDNOT 602.14  ; #3腔体平移一级气缸缩回[A]
AND 803.03  ; #3腔体顶伸气缸下降位标志[0003.03]
AND W4.04  ; 初次上电#3腔体平移一级气缸伸出条件
ANDNOT A281.05  ; 进料伺服Z轴无原点标志(0：原点确定,1：原点未确定)
AND H24.01  ; 进料伺服Z轴回原点记Z忆
AND 851.03  ; 进料伺服Z轴待机位标志
ANDNOT A327.05  ; 出料伺服Z轴无原点标志(0：原点确定,1：原点未确定)
AND 853.03  ; 出料伺服Z轴待机位标志
ORLD
ANDLD
SET 12.15  ; #3腔体平移一级气缸伸出
RSET 12.14  ; #3腔体平移一级气缸缩回
LD TR0
AND P_First_Cycle
AND P_On
SET W4.04  ; 初次上电#3腔体平移一级气缸伸出条件
LD TR0
LD 402.14  ; #3腔体平移一级气缸缩回[M]
OR 602.14  ; #3腔体平移一级气缸缩回[A]
OR 12.15  ; #3腔体平移一级气缸伸出
OR W1.01  ; 自动模式
ANDLD
RSET W4.04  ; 初次上电#3腔体平移一级气缸伸出条件

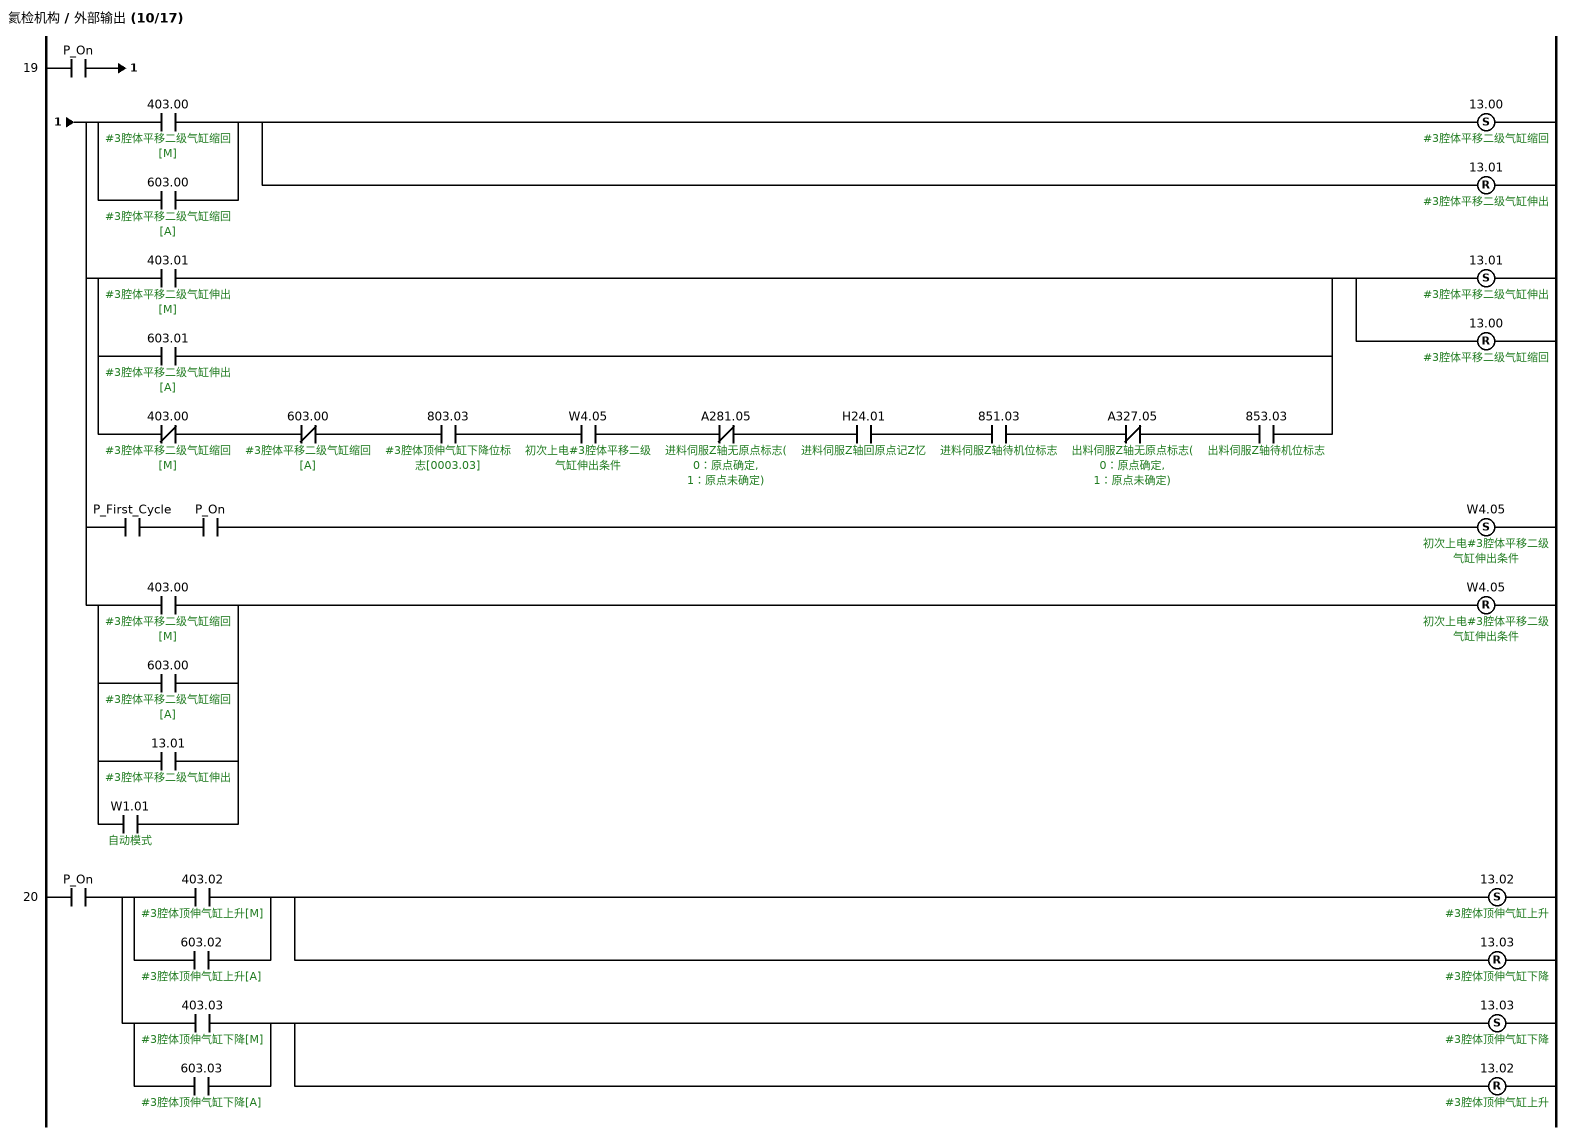
; rung 19
LD P_On
OUT TR0
LD 403.00  ; #3腔体平移二级气缸缩回[M]
OR 603.00  ; #3腔体平移二级气缸缩回[A]
ANDLD
SET 13.00  ; #3腔体平移二级气缸缩回
RSET 13.01  ; #3腔体平移二级气缸伸出
LD TR0
LD 403.01  ; #3腔体平移二级气缸伸出[M]
OR 603.01  ; #3腔体平移二级气缸伸出[A]
LDNOT 403.00  ; #3腔体平移二级气缸缩回[M]
ANDNOT 603.00  ; #3腔体平移二级气缸缩回[A]
AND 803.03  ; #3腔体顶伸气缸下降位标志[0003.03]
AND W4.05  ; 初次上电#3腔体平移二级气缸伸出条件
ANDNOT A281.05  ; 进料伺服Z轴无原点标志(0：原点确定,1：原点未确定)
AND H24.01  ; 进料伺服Z轴回原点记Z忆
AND 851.03  ; 进料伺服Z轴待机位标志
ANDNOT A327.05  ; 出料伺服Z轴无原点标志(0：原点确定,1：原点未确定)
AND 853.03  ; 出料伺服Z轴待机位标志
ORLD
ANDLD
SET 13.01  ; #3腔体平移二级气缸伸出
RSET 13.00  ; #3腔体平移二级气缸缩回
LD TR0
AND P_First_Cycle
AND P_On
SET W4.05  ; 初次上电#3腔体平移二级气缸伸出条件
LD TR0
LD 403.00  ; #3腔体平移二级气缸缩回[M]
OR 603.00  ; #3腔体平移二级气缸缩回[A]
OR 13.01  ; #3腔体平移二级气缸伸出
OR W1.01  ; 自动模式
ANDLD
RSET W4.05  ; 初次上电#3腔体平移二级气缸伸出条件
; rung 20
LD P_On
OUT TR0
LD 403.02  ; #3腔体顶伸气缸上升[M]
OR 603.02  ; #3腔体顶伸气缸上升[A]
ANDLD
SET 13.02  ; #3腔体顶伸气缸上升
RSET 13.03  ; #3腔体顶伸气缸下降
LD TR0
LD 403.03  ; #3腔体顶伸气缸下降[M]
OR 603.03  ; #3腔体顶伸气缸下降[A]
ANDLD
SET 13.03  ; #3腔体顶伸气缸下降
RSET 13.02  ; #3腔体顶伸气缸上升

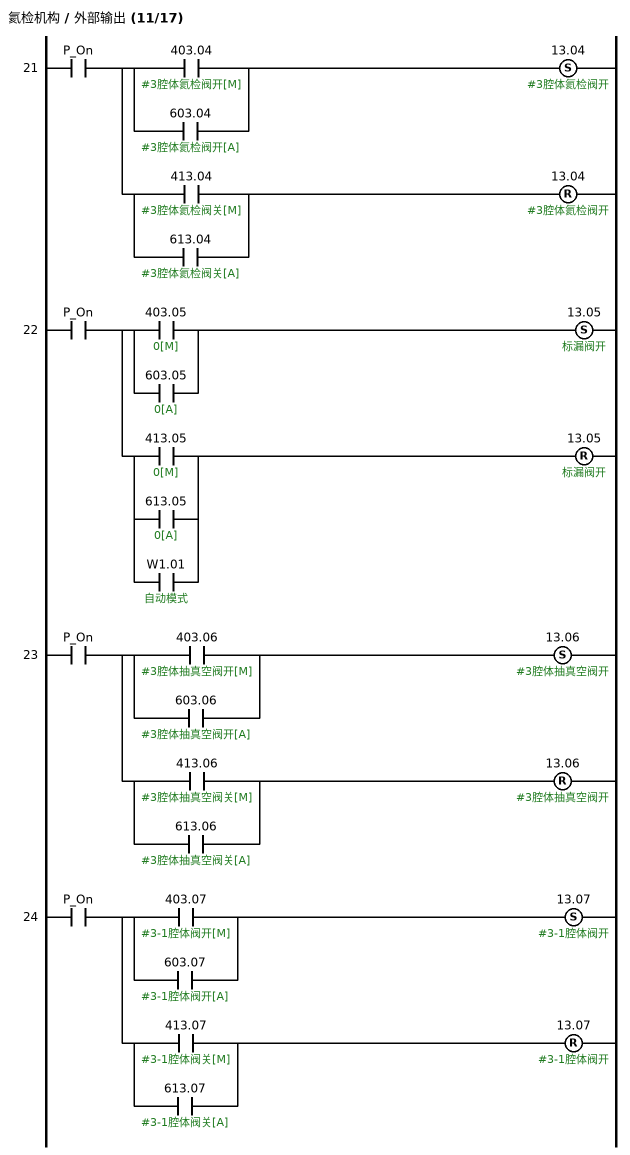
; rung 21
LD P_On
OUT TR0
LD 403.04  ; #3腔体氦检阀开[M]
OR 603.04  ; #3腔体氦检阀开[A]
ANDLD
SET 13.04  ; #3腔体氦检阀开
LD TR0
LD 413.04  ; #3腔体氦检阀关[M]
OR 613.04  ; #3腔体氦检阀关[A]
ANDLD
RSET 13.04  ; #3腔体氦检阀开
; rung 22
LD P_On
OUT TR0
LD 403.05  ; 0[M]
OR 603.05  ; 0[A]
ANDLD
SET 13.05  ; 标漏阀开
LD TR0
LD 413.05  ; 0[M]
OR 613.05  ; 0[A]
OR W1.01  ; 自动模式
ANDLD
RSET 13.05  ; 标漏阀开
; rung 23
LD P_On
OUT TR0
LD 403.06  ; #3腔体抽真空阀开[M]
OR 603.06  ; #3腔体抽真空阀开[A]
ANDLD
SET 13.06  ; #3腔体抽真空阀开
LD TR0
LD 413.06  ; #3腔体抽真空阀关[M]
OR 613.06  ; #3腔体抽真空阀关[A]
ANDLD
RSET 13.06  ; #3腔体抽真空阀开
; rung 24
LD P_On
OUT TR0
LD 403.07  ; #3-1腔体阀开[M]
OR 603.07  ; #3-1腔体阀开[A]
ANDLD
SET 13.07  ; #3-1腔体阀开
LD TR0
LD 413.07  ; #3-1腔体阀关[M]
OR 613.07  ; #3-1腔体阀关[A]
ANDLD
RSET 13.07  ; #3-1腔体阀开

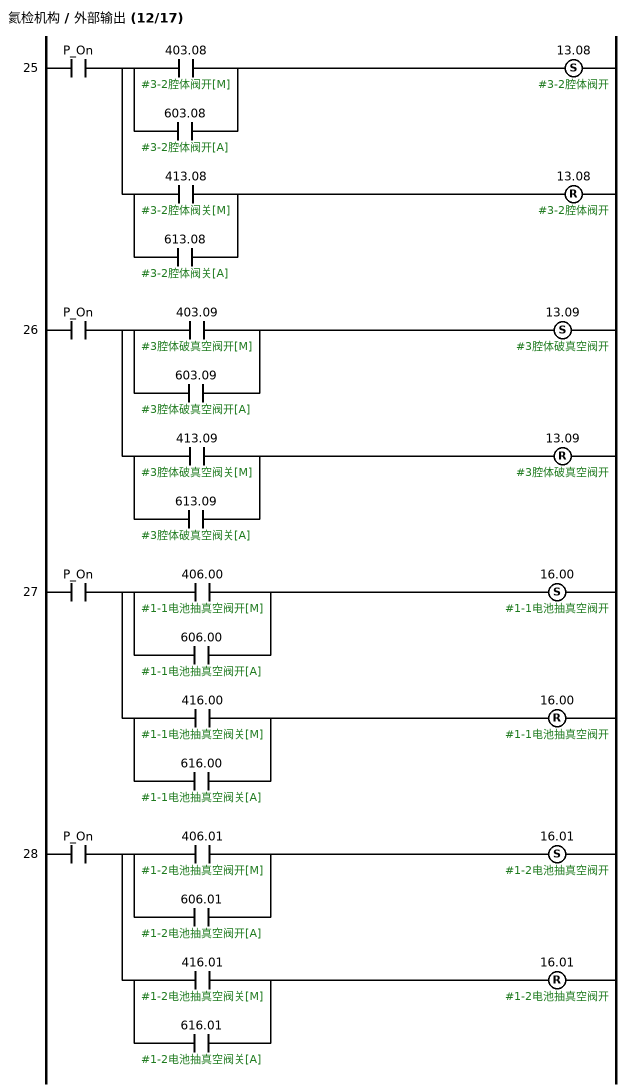
; rung 25
LD P_On
OUT TR0
LD 403.08  ; #3-2腔体阀开[M]
OR 603.08  ; #3-2腔体阀开[A]
ANDLD
SET 13.08  ; #3-2腔体阀开
LD TR0
LD 413.08  ; #3-2腔体阀关[M]
OR 613.08  ; #3-2腔体阀关[A]
ANDLD
RSET 13.08  ; #3-2腔体阀开
; rung 26
LD P_On
OUT TR0
LD 403.09  ; #3腔体破真空阀开[M]
OR 603.09  ; #3腔体破真空阀开[A]
ANDLD
SET 13.09  ; #3腔体破真空阀开
LD TR0
LD 413.09  ; #3腔体破真空阀关[M]
OR 613.09  ; #3腔体破真空阀关[A]
ANDLD
RSET 13.09  ; #3腔体破真空阀开
; rung 27
LD P_On
OUT TR0
LD 406.00  ; #1-1电池抽真空阀开[M]
OR 606.00  ; #1-1电池抽真空阀开[A]
ANDLD
SET 16.00  ; #1-1电池抽真空阀开
LD TR0
LD 416.00  ; #1-1电池抽真空阀关[M]
OR 616.00  ; #1-1电池抽真空阀关[A]
ANDLD
RSET 16.00  ; #1-1电池抽真空阀开
; rung 28
LD P_On
OUT TR0
LD 406.01  ; #1-2电池抽真空阀开[M]
OR 606.01  ; #1-2电池抽真空阀开[A]
ANDLD
SET 16.01  ; #1-2电池抽真空阀开
LD TR0
LD 416.01  ; #1-2电池抽真空阀关[M]
OR 616.01  ; #1-2电池抽真空阀关[A]
ANDLD
RSET 16.01  ; #1-2电池抽真空阀开

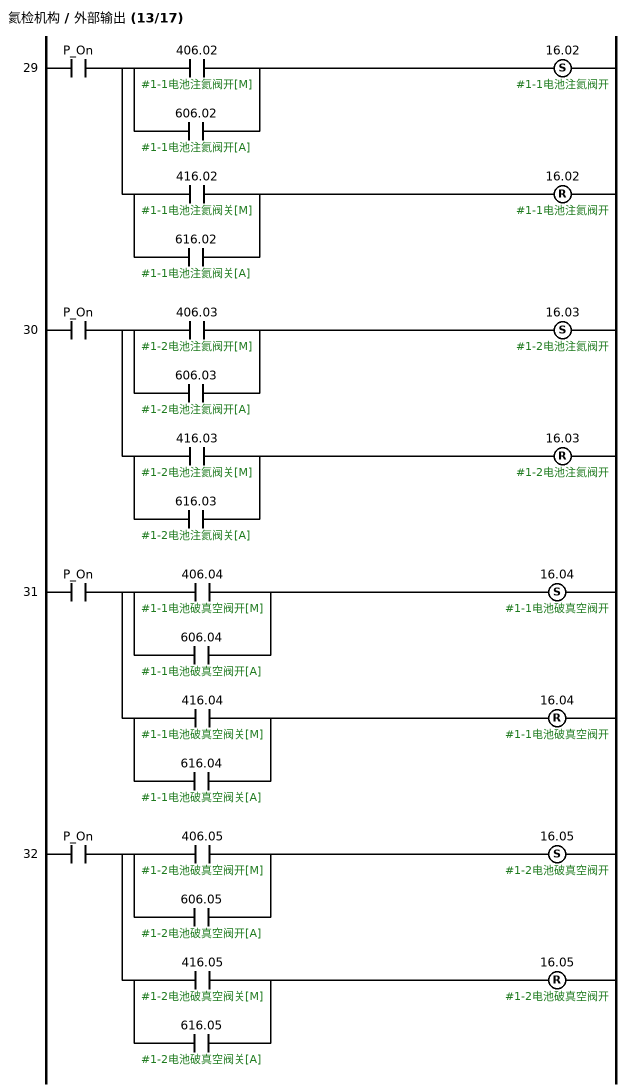
; rung 29
LD P_On
OUT TR0
LD 406.02  ; #1-1电池注氦阀开[M]
OR 606.02  ; #1-1电池注氦阀开[A]
ANDLD
SET 16.02  ; #1-1电池注氦阀开
LD TR0
LD 416.02  ; #1-1电池注氦阀关[M]
OR 616.02  ; #1-1电池注氦阀关[A]
ANDLD
RSET 16.02  ; #1-1电池注氦阀开
; rung 30
LD P_On
OUT TR0
LD 406.03  ; #1-2电池注氦阀开[M]
OR 606.03  ; #1-2电池注氦阀开[A]
ANDLD
SET 16.03  ; #1-2电池注氦阀开
LD TR0
LD 416.03  ; #1-2电池注氦阀关[M]
OR 616.03  ; #1-2电池注氦阀关[A]
ANDLD
RSET 16.03  ; #1-2电池注氦阀开
; rung 31
LD P_On
OUT TR0
LD 406.04  ; #1-1电池破真空阀开[M]
OR 606.04  ; #1-1电池破真空阀开[A]
ANDLD
SET 16.04  ; #1-1电池破真空阀开
LD TR0
LD 416.04  ; #1-1电池破真空阀关[M]
OR 616.04  ; #1-1电池破真空阀关[A]
ANDLD
RSET 16.04  ; #1-1电池破真空阀开
; rung 32
LD P_On
OUT TR0
LD 406.05  ; #1-2电池破真空阀开[M]
OR 606.05  ; #1-2电池破真空阀开[A]
ANDLD
SET 16.05  ; #1-2电池破真空阀开
LD TR0
LD 416.05  ; #1-2电池破真空阀关[M]
OR 616.05  ; #1-2电池破真空阀关[A]
ANDLD
RSET 16.05  ; #1-2电池破真空阀开

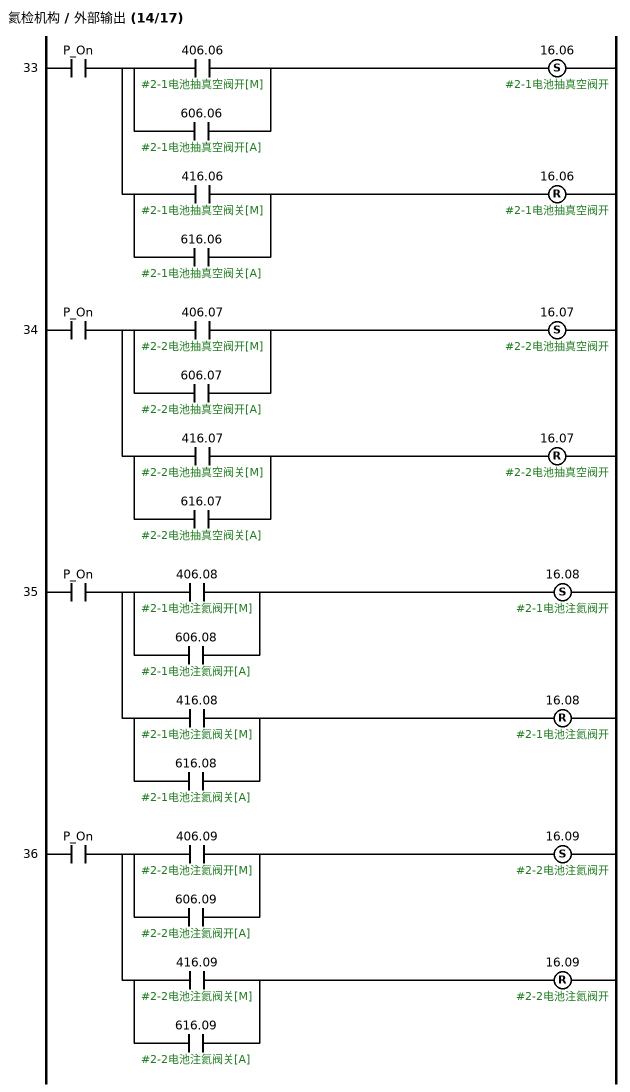
; rung 33
LD P_On
OUT TR0
LD 406.06  ; #2-1电池抽真空阀开[M]
OR 606.06  ; #2-1电池抽真空阀开[A]
ANDLD
SET 16.06  ; #2-1电池抽真空阀开
LD TR0
LD 416.06  ; #2-1电池抽真空阀关[M]
OR 616.06  ; #2-1电池抽真空阀关[A]
ANDLD
RSET 16.06  ; #2-1电池抽真空阀开
; rung 34
LD P_On
OUT TR0
LD 406.07  ; #2-2电池抽真空阀开[M]
OR 606.07  ; #2-2电池抽真空阀开[A]
ANDLD
SET 16.07  ; #2-2电池抽真空阀开
LD TR0
LD 416.07  ; #2-2电池抽真空阀关[M]
OR 616.07  ; #2-2电池抽真空阀关[A]
ANDLD
RSET 16.07  ; #2-2电池抽真空阀开
; rung 35
LD P_On
OUT TR0
LD 406.08  ; #2-1电池注氦阀开[M]
OR 606.08  ; #2-1电池注氦阀开[A]
ANDLD
SET 16.08  ; #2-1电池注氦阀开
LD TR0
LD 416.08  ; #2-1电池注氦阀关[M]
OR 616.08  ; #2-1电池注氦阀关[A]
ANDLD
RSET 16.08  ; #2-1电池注氦阀开
; rung 36
LD P_On
OUT TR0
LD 406.09  ; #2-2电池注氦阀开[M]
OR 606.09  ; #2-2电池注氦阀开[A]
ANDLD
SET 16.09  ; #2-2电池注氦阀开
LD TR0
LD 416.09  ; #2-2电池注氦阀关[M]
OR 616.09  ; #2-2电池注氦阀关[A]
ANDLD
RSET 16.09  ; #2-2电池注氦阀开

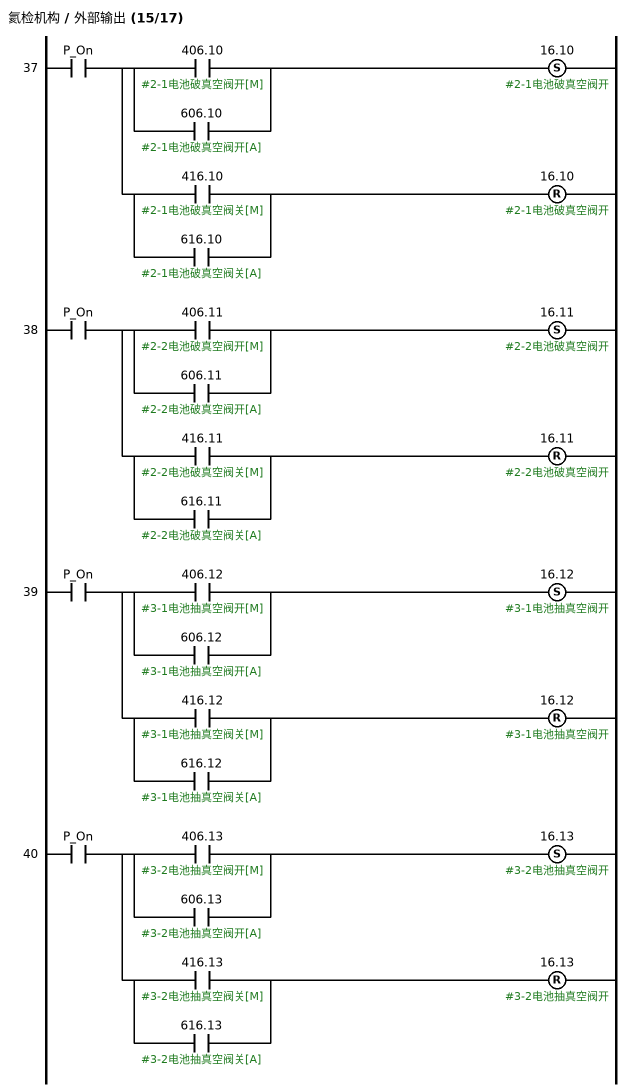
; rung 37
LD P_On
OUT TR0
LD 406.10  ; #2-1电池破真空阀开[M]
OR 606.10  ; #2-1电池破真空阀开[A]
ANDLD
SET 16.10  ; #2-1电池破真空阀开
LD TR0
LD 416.10  ; #2-1电池破真空阀关[M]
OR 616.10  ; #2-1电池破真空阀关[A]
ANDLD
RSET 16.10  ; #2-1电池破真空阀开
; rung 38
LD P_On
OUT TR0
LD 406.11  ; #2-2电池破真空阀开[M]
OR 606.11  ; #2-2电池破真空阀开[A]
ANDLD
SET 16.11  ; #2-2电池破真空阀开
LD TR0
LD 416.11  ; #2-2电池破真空阀关[M]
OR 616.11  ; #2-2电池破真空阀关[A]
ANDLD
RSET 16.11  ; #2-2电池破真空阀开
; rung 39
LD P_On
OUT TR0
LD 406.12  ; #3-1电池抽真空阀开[M]
OR 606.12  ; #3-1电池抽真空阀开[A]
ANDLD
SET 16.12  ; #3-1电池抽真空阀开
LD TR0
LD 416.12  ; #3-1电池抽真空阀关[M]
OR 616.12  ; #3-1电池抽真空阀关[A]
ANDLD
RSET 16.12  ; #3-1电池抽真空阀开
; rung 40
LD P_On
OUT TR0
LD 406.13  ; #3-2电池抽真空阀开[M]
OR 606.13  ; #3-2电池抽真空阀开[A]
ANDLD
SET 16.13  ; #3-2电池抽真空阀开
LD TR0
LD 416.13  ; #3-2电池抽真空阀关[M]
OR 616.13  ; #3-2电池抽真空阀关[A]
ANDLD
RSET 16.13  ; #3-2电池抽真空阀开

